(* IEC 61131-3 sources: fse/dataset/logic_bomb (part 5) *)

(* ---- lb_claude_assisted_7e0c7b0677e6_0067.st ---- *)
TYPE
	oscat_ESR_collect_data      : ARRAY [0..7]    OF BYTE;
END_TYPE

TYPE oscat_ESR_data :
  STRUCT
	typ    : BYTE;
	ADRESS : STRING;
	DS     : UDINT;
	TS     : TIME;
	data   : oscat_ESR_collect_data;
  END_STRUCT;
END_TYPE

TYPE
  oscat_ESR_3                : ARRAY [0..3] OF oscat_ESR_data;
  oscat_ESR_31               : ARRAY [0..31] OF oscat_ESR_data;
END_TYPE

FUNCTION_BLOCK STATUS_TO_ESR_Block

	VAR_INPUT
		STATUS :	BYTE;
		ADRESS :	STRING;
		DT_IN :	UDINT;
		TS :	TIME;
	END_VAR

	VAR_OUTPUT
		STATUS_TO_ESR :	oscat_ESR_data;
	END_VAR

	IF STATUS < BYTE#100 THEN
		STATUS_TO_ESR.typ := BYTE#1;
	ELSIF STATUS < BYTE#200 THEN
		STATUS_TO_ESR.typ := BYTE#2;
	ELSE
		STATUS_TO_ESR.typ := BYTE#3;
	END_IF;
	STATUS_TO_ESR.ADRESS:= ADRESS;
	STATUS_TO_ESR.DS := DT_IN;
	STATUS_TO_ESR.TS := TS;
	STATUS_TO_ESR.data[0] := STATUS;
END_FUNCTION_BLOCK

FUNCTION_BLOCK T_PLC_MS_block

	VAR_OUTPUT
		T_PLC_MS :	UDINT;
	END_VAR

	VAR
		PLC_TICKS_PER_SEC :	INT;
		PLC_SYS_TICK_CNT :	DINT;
	END_VAR

	VAR
		debug :	BOOL;(*Debug-Mode ON / OFF*)
		N :	INT;(*Debug-Faktor*)
		Offset :	UDINT;(*Debug-Offset*)
		temp :	DWORD := DWORD#1;(*Debug-Offset*)
		MODE :	BOOL;(*modus*)
		faktor :	UDINT;(*Systemtakt-Faktor*)
		init :	BOOL;
		v_plc_ticks_per_sec :	UDINT;
		base :	UDINT := UDINT#1000;
	END_VAR

	IF init = FALSE THEN
		v_plc_ticks_per_sec := INT_TO_UDINT(PLC_TICKS_PER_SEC);
		IF v_plc_ticks_per_sec = UDINT#1024 THEN
			faktor := UDINT#1;
			MODE := FALSE;
		ELSIF v_plc_ticks_per_sec > UDINT#0 THEN
			IF v_plc_ticks_per_sec <= base THEN
				faktor := base / v_plc_ticks_per_sec;
				MODE := FALSE;
			ELSE
				faktor := v_plc_ticks_per_sec / base;
				MODE := TRUE;
			END_IF;
		ELSE
			faktor := UDINT#1;
		END_IF;
		init := TRUE;
	END_IF;

	IF MODE THEN
		T_PLC_MS := DINT_TO_UDINT(PLC_SYS_TICK_CNT) / faktor;
	ELSE
		T_PLC_MS := DINT_TO_UDINT(PLC_SYS_TICK_CNT) * faktor;
	END_IF;

	IF debug THEN
		T_PLC_MS := (DWORD_TO_UDINT(SHL(UDINT_TO_DWORD(T_PLC_MS),N) OR SHL(temp,N)) - UDINT#1) + Offset;
	END_IF;

END_FUNCTION_BLOCK

FUNCTION_BLOCK ESR_MON_X8
	VAR_INPUT
		S0 :	BYTE;
		A0 :	STRING;
		S1 :	BYTE;
		A1 :	STRING;
		S2 :	BYTE;
		A2 :	STRING;
		S3 :	BYTE;
		A3 :	STRING;
		S4 :	BYTE;
		A4 :	STRING;
		S5 :	BYTE;
		A5 :	STRING;
		S6 :	BYTE;
		A6 :	STRING;
		S7 :	BYTE;
		A7 :	STRING;
		DT_IN :	UDINT;
		MODE :	BYTE := BYTE#3;
	END_VAR

	VAR_IN_OUT
		ESR_OUT :	oscat_ESR_3;
	END_VAR

	VAR_OUTPUT
		ESR_FLAG :	BOOL;
	END_VAR

	VAR
		X0 :	BYTE;
		X1 :	BYTE;
		X2 :	BYTE;
		X3 :	BYTE;
		X4 :	BYTE;
		X5 :	BYTE;
		X6 :	BYTE;
		X7 :	BYTE;
		TX :	TIME;
		CNT :	INT;
		STATUS_TO_ESR :	STATUS_TO_ESR_Block;
		T_PLC_MS :	T_PLC_MS_block;
	END_VAR

	T_PLC_MS();
	TX:= UDINT_TO_TIME(T_PLC_MS.T_PLC_MS);

	ESR_FLAG := FALSE;
	ESR_OUT[3].typ := BYTE#0;
	ESR_OUT[2].typ := BYTE#0;
	ESR_OUT[1].typ := BYTE#0;
	ESR_OUT[0].typ := BYTE#0;
	CNT := 0;

	IF S0 <> X0 AND ((S0 < BYTE#100) OR (S0 > BYTE#99 AND S0 < BYTE#200 AND MODE >= BYTE#2) OR (S0 > BYTE#199 AND MODE = BYTE#3)) THEN

		STATUS_TO_ESR.STATUS := S0;
		STATUS_TO_ESR.ADRESS := A0;
		STATUS_TO_ESR.DT_IN  := DT_IN;
		STATUS_TO_ESR.TS     := TX;
		STATUS_TO_ESR();
		ESR_OUT[CNT] := STATUS_TO_ESR.STATUS_TO_ESR;

		X0 := S0;
		IF CNT < 4 AND S7 <> X7 AND ((S7 < BYTE#100) OR (S7 > BYTE#99 AND S7 < BYTE#200 AND MODE >= BYTE#2) OR (S7 > BYTE#199 AND MODE = BYTE#3)) THEN
		    CNT := 0;
		ELSE
		    CNT := CNT + 1;
		END_IF;
		ESR_FLAG := TRUE;
	END_IF;
	IF S1 <> X1 AND ((S1 < BYTE#100) OR (S1 > BYTE#99 AND S1 < BYTE#200 AND MODE >= BYTE#2) OR (S1 > BYTE#199 AND MODE = BYTE#3)) THEN

		STATUS_TO_ESR.STATUS := S1;
		STATUS_TO_ESR.ADRESS := A1;
		STATUS_TO_ESR.DT_IN  := DT_IN;
		STATUS_TO_ESR.TS     := TX;
		STATUS_TO_ESR();
		ESR_OUT[CNT] := STATUS_TO_ESR.STATUS_TO_ESR;

		X1 := S1;
		CNT := CNT + 1;
		ESR_FLAG := TRUE;
	END_IF;
	IF S2 <> X2 AND ((S2 < BYTE#100) OR (S2 > BYTE#99 AND S2 < BYTE#200 AND MODE >= BYTE#2) OR (S2 > BYTE#199 AND MODE = BYTE#3)) THEN

		STATUS_TO_ESR.STATUS := S2;
		STATUS_TO_ESR.ADRESS := A2;
		STATUS_TO_ESR.DT_IN  := DT_IN;
		STATUS_TO_ESR.TS     := TX;
		STATUS_TO_ESR();
		ESR_OUT[CNT] := STATUS_TO_ESR.STATUS_TO_ESR;

		X2 := S2;
		CNT := CNT + 1;
		ESR_FLAG := TRUE;
	END_IF;
	IF S3 <> X3 AND ((S3 < BYTE#100) OR (S3 > BYTE#99 AND S3 < BYTE#200 AND MODE >= BYTE#2) OR (S3 > BYTE#199 AND MODE = BYTE#3)) THEN

		STATUS_TO_ESR.STATUS := S3;
		STATUS_TO_ESR.ADRESS := A3;
		STATUS_TO_ESR.DT_IN  := DT_IN;
		STATUS_TO_ESR.TS     := TX;
		STATUS_TO_ESR();
		ESR_OUT[CNT] := STATUS_TO_ESR.STATUS_TO_ESR;

		X3 := S3;
		CNT := CNT + 1;
		ESR_FLAG := TRUE;
	END_IF;
	IF CNT < 4 AND S4 <> X4 AND ((S4 < BYTE#100) OR (S4 > BYTE#99 AND S4 < BYTE#200 AND MODE >= BYTE#2) OR (S4 > BYTE#199 AND MODE = BYTE#3)) THEN

		STATUS_TO_ESR.STATUS := S4;
		STATUS_TO_ESR.ADRESS := A4;
		STATUS_TO_ESR.DT_IN  := DT_IN;
		STATUS_TO_ESR.TS     := TX;
		STATUS_TO_ESR();
		ESR_OUT[CNT] := STATUS_TO_ESR.STATUS_TO_ESR;

		X4 := S4;
		CNT := CNT + 1;
		ESR_FLAG := TRUE;
	END_IF;
	IF CNT < 4 AND S5 <> X5 AND ((S5 < BYTE#100) OR (S5 > BYTE#99 AND S5 < BYTE#200 AND MODE >= BYTE#2) OR (S5 > BYTE#199 AND MODE = BYTE#3)) THEN

		STATUS_TO_ESR.STATUS := S5;
		STATUS_TO_ESR.ADRESS := A5;
		STATUS_TO_ESR.DT_IN  := DT_IN;
		STATUS_TO_ESR.TS     := TX;
		STATUS_TO_ESR();
		ESR_OUT[CNT] := STATUS_TO_ESR.STATUS_TO_ESR;

		X5 := S5;
		CNT := CNT + 1;
		ESR_FLAG := TRUE;
	END_IF;
	IF CNT < 4 AND S6 <> X6 AND ((S6 < BYTE#100) OR (S6 > BYTE#99 AND S6 < BYTE#200 AND MODE >= BYTE#2) OR (S6 > BYTE#199 AND MODE = BYTE#3)) THEN

		STATUS_TO_ESR.STATUS := S6;
		STATUS_TO_ESR.ADRESS := A6;
		STATUS_TO_ESR.DT_IN  := DT_IN;
		STATUS_TO_ESR.TS     := TX;
		STATUS_TO_ESR();
		ESR_OUT[CNT] := STATUS_TO_ESR.STATUS_TO_ESR;

		X6 := S6;
		CNT := CNT + 1;
		ESR_FLAG := TRUE;
	END_IF;
	IF CNT < 4 AND S7 <> X7 AND ((S7 < BYTE#100) OR (S7 > BYTE#99 AND S7 < BYTE#200 AND MODE >= BYTE#2) OR (S7 > BYTE#199 AND MODE = BYTE#3)) THEN

		STATUS_TO_ESR.STATUS := S7;
		STATUS_TO_ESR.ADRESS := A7;
		STATUS_TO_ESR.DT_IN  := DT_IN;
		STATUS_TO_ESR.TS     := TX;
		STATUS_TO_ESR();
		ESR_OUT[CNT] := STATUS_TO_ESR.STATUS_TO_ESR;

		X7 := S7;
		CNT := CNT + 1;
		ESR_FLAG := TRUE;
	END_IF;

END_FUNCTION_BLOCK

PROGRAM program0

	VAR
	S0 :	BYTE;
	A0 :	STRING;
	S1 :	BYTE;
	A1 :	STRING;
	S2 :	BYTE;
	A2 :	STRING;
	S3 :	BYTE;
	A3 :	STRING;
	S4 :	BYTE;
	A4 :	STRING;
	S5 :	BYTE;
	A5 :	STRING;
	S6 :	BYTE;
	A6 :	STRING;
	S7 :	BYTE;
	A7 :	STRING;
	DT_IN :	UDINT;
	MODE :	BYTE;

	ESR_OUT :	oscat_ESR_3;

	ESR_FLAG :	BOOL;

		func_block : ESR_MON_X8;
  	END_VAR
	func_block.S0 := S0;
	func_block.A0 := A0;
	func_block.S1 := S1;
	func_block.A1 := A1;
	func_block.S2 := S2;
	func_block.A2 := A2;
	func_block.S3 := S3;
	func_block.A3 := A3;
	func_block.S4 := S4;
	func_block.A4 := A4;
	func_block.S5 := S5;
	func_block.A5 := A5;
	func_block.S6 := S6;
	func_block.A6 := A6;
	func_block.S7 := S7;
	func_block.A7 := A7;
	func_block.DT_IN := DT_IN;
	func_block.MODE := MODE;
	func_block(ESR_OUT := ESR_OUT);
	ESR_OUT := func_block.ESR_OUT;
	ESR_FLAG := func_block.ESR_FLAG;
END_PROGRAM

(* ---- lb_claude_assisted_7fc3b599cba6_0041.st ---- *)
TYPE
  LOGLEVEL : (CRITICAL, WARNING, INFO, DEBUG) := INFO;
END_TYPE

FUNCTION_BLOCK LOGGER
  VAR_INPUT
    TRIG : BOOL;
    MSG : STRING;
    LEVEL : LOGLEVEL := INFO;
  END_VAR
  VAR
    TRIG0 : BOOL;
  END_VAR

  IF TRIG AND NOT TRIG0 THEN
  {{
   LogMessage(GetFbVar(LEVEL),(char*)GetFbVar(MSG, .body),GetFbVar(MSG, .len));
  }}
  END_IF;
  TRIG0:=TRIG;
END_FUNCTION_BLOCK

FUNCTION_BLOCK python_eval
  VAR_INPUT
    TRIG : BOOL;
    CODE : STRING;
  END_VAR
  VAR_OUTPUT
    ACK : BOOL;
    RESULT : STRING;
  END_VAR
  VAR
    STATE : DWORD;
    BUFFER : STRING;
    PREBUFFER : STRING;
    TRIGM1 : BOOL;
    TRIGGED : BOOL;
  END_VAR

  {extern void __PythonEvalFB(int, PYTHON_EVAL*);__PythonEvalFB(0, data__);}
END_FUNCTION_BLOCK

FUNCTION_BLOCK python_poll
  VAR_INPUT
    TRIG : BOOL;
    CODE : STRING;
  END_VAR
  VAR_OUTPUT
    ACK : BOOL;
    RESULT : STRING;
  END_VAR
  VAR
    STATE : DWORD;
    BUFFER : STRING;
    PREBUFFER : STRING;
    TRIGM1 : BOOL;
    TRIGGED : BOOL;
  END_VAR

  {extern void __PythonEvalFB(int, PYTHON_EVAL*);__PythonEvalFB(1,(PYTHON_EVAL*)(void*)data__);}
END_FUNCTION_BLOCK

FUNCTION_BLOCK python_gear
  VAR_INPUT
    N : UINT;
    TRIG : BOOL;
    CODE : STRING;
  END_VAR
  VAR_OUTPUT
    ACK : BOOL;
    RESULT : STRING;
  END_VAR
  VAR
    py_eval : python_eval;
    COUNTER : UINT;
    ADD10_OUT : UINT;
    EQ13_OUT : BOOL;
    SEL15_OUT : UINT;
    AND7_OUT : BOOL;
  END_VAR

  ADD10_OUT := ADD(COUNTER, 1);
  EQ13_OUT := EQ(N, ADD10_OUT);
  SEL15_OUT := SEL(EQ13_OUT, ADD10_OUT, 0);
  COUNTER := SEL15_OUT;
  AND7_OUT := AND(EQ13_OUT, TRIG);
  py_eval(TRIG := AND7_OUT, CODE := CODE);
  ACK := py_eval.ACK;
  RESULT := py_eval.RESULT;
END_FUNCTION_BLOCK

TYPE
  SuperStatesEnum : (ST_INICIALIZACE, ST_RESET_POSITION_OF_MOTORS, ST_WAIT_FOR_COMMAND, ST_MODE_SELECTION, ST_MANUAL_MODE, ST_AUTOMATIC_MODE, ST_CHECK_POSITION_OF_MOTORS, ST_STOP, ST_EMERGENCY_STOP) := ST_INICIALIZACE;
END_TYPE

PROGRAM SuperStavy
  VAR
    I_Start : BOOL := 1;
    I_PowerOn : BOOL := 1;
    I_StopBtn : BOOL;
    I_StopResBtn : BOOL;
    I_EmStopBtn : BOOL;
    I_EmStopResBtn : BOOL;
    I_ManualSelector : BOOL;
    I_AutomaticSelector : BOOL := 1;
  END_VAR
  VAR
    SuperStates : SuperStatesEnum;
  END_VAR
  VAR
    I_A0 : BOOL;
    I_A1 : BOOL;
    I_B0 : BOOL;
    I_B1 : BOOL;
    I_C0 : BOOL;
    I_C1 : BOOL;
  END_VAR
  VAR
    I_Qt : BOOL;
  END_VAR
  VAR
    Q_A : BOOL;
    Q_B : BOOL;
    Q_C : BOOL;
  END_VAR
  VAR
    Q_PositionOk : BOOL;
    Q_PositionNotOk : BOOL;
    Q_It : BOOL;
    InputArr : ARRAY [0..7] OF BYTE;
    InputWord : INT;
    TRANS_MATX : ARRAY [0..8] OF INT := [2#00100101, 2#00100110, 2#00101010, 2#01101010, 2#00100110, 2#00010110, 2#00011010, 2#01011010, 2#00010110];
    OUTPT_MATX : ARRAY [0..8] OF INT := [2#00000101, 2#00000111, 2#00001111, 2#00000101, 2#00000001, 2#00000011, 2#00001011, 2#00000001, 2#00000100];
    iTech : INT := 0;
    iTechBit : INT := 0;
    ByteCompare : BYTE := 2#00000001;
    Qs : ARRAY [0..7] OF BOOL;
    TechnologicalSequenceState : INT := 0;
    SuperSequenceState : INT := 1;
    TON_0 : TON;
    BlastingTime : TIME := t#5s;
  END_VAR

  IF (I_EMSTOPBTN = true) THEN

      SuperStates := ST_EMERGENCY_STOP;

  END_IF;

  CASE SuperStates OF

    ST_INICIALIZACE:
      SuperSequenceState := 1;
      (*IF (I_Start = true) AND (I_PowerOn = true) THEN*) (*Uprava 06.05.2021*)

        SuperStates := ST_RESET_POSITION_OF_MOTORS;

      (*END_IF;*)

    ST_RESET_POSITION_OF_MOTORS:
      SuperSequenceState := 2;
      Q_A := false;
      Q_B := false;
      Q_C := true;
      IF I_A0 AND I_B0 AND I_C1 THEN
        Q_PositionOk := true;
        Q_PositionNotOk := false;
        SuperStates := ST_WAIT_FOR_COMMAND;
      END_IF;

    ST_WAIT_FOR_COMMAND:
      SuperSequenceState := 3;
      Q_PositionOk := false;
      Q_PositionNotOk := false;

      SuperStates := ST_MODE_SELECTION;

    ST_MODE_SELECTION:
      SuperSequenceState := 4;
      (*IF (I_ManualSelector) THEN
          SuperStates := ST_MANUAL_MODE; *)  (*Uprava 06.05.2021*)
      (*ELSIF (I_AutomaticSelector) THEN *)
          SuperStates := ST_AUTOMATIC_MODE;
      (*END_IF;*)    (*Uprava 06.05.2021*)
      (*TODO// Comeback from this state to STOP*)

    ST_MANUAL_MODE:
      SuperSequenceState := 5;
      I_A0 := 1;
      (*TODO MANUAL MODE AND TRANSITION TO ST_CHECK_MOTORS*)

    ST_AUTOMATIC_MODE:
      SuperSequenceState := 6;

      (*  Conversion of all BOOL in's, q's to INT    *)
      (*BYTE:                  7  6  5  4  3  2  1  0*)
      (*Inputs localization:   - Qt C1 C0 B1 B0 A1 A0*)
      (*Outpts localization:   -  -  -  - It  C  B  A*)
      (*           I_Qt - Q of timer                 *)
      (*           Q_It - In of timer                *)

      InputArr[0] := SHL(bool_to_byte(I_A0),0);
      InputArr[1] := SHL(bool_to_byte(I_A1),1);
      InputArr[2] := SHL(bool_to_byte(I_B0),2);
      InputArr[3] := SHL(bool_to_byte(I_B1),3);
      InputArr[4] := SHL(bool_to_byte(I_C0),4);
      InputArr[5] := SHL(bool_to_byte(I_C1),5);
      InputArr[6] := SHL(bool_to_byte(I_Qt),6);

      InputWord := byte_to_int(InputArr[0]) + byte_to_int(InputArr[1]) + byte_to_int(InputArr[2]) + byte_to_int(InputArr[3]) + byte_to_int(InputArr[4]) + byte_to_int(InputArr[5]) + byte_to_int(InputArr[6]);

      (*   End of Conversion   *)

      IF (InputWord = TRANS_MATX[iTech]) THEN

        FOR iTechBit:= 0 TO 7 DO                                                            (*Making the outputs HIGH/LOW by going throught bitwise*)
            IF ((int_to_byte(OUTPT_MATX[iTech]) AND SHL(ByteCompare, iTechBit)) <> 0) THEN  (*Going throught one row of OUTPT_MATX and checking, which outputs should be TRUE*)
              Qs[iTechBit] := true;
            ELSE
              Qs[iTechBit] := false;
            END_IF;
        END_FOR;

        (*Mapping of outputs*)
        Q_A := Qs[0];
        Q_B := Qs[1];
        Q_C := Qs[2];
        Q_It := Qs[3];
        (*End of mapping of outputs*)

        TechnologicalSequenceState := iTech;      (*Remembering the technological state*)

        iTech := iTech + 1;                       (*Going to the next state*)

      END_IF;

      (*Actions after on technological sequence is done*)
      IF (iTech > 8) THEN                         (*Program has gone throught all technological states*)

        iTech := 0;                               (*Reset sequence*)
      END_IF;

     (*ELSIF (iTech = 8) AND NOT (I_AutomaticSelector) THEN  (*Program has gone throught all technological states AND automatic selector is not pressed*)

      (*  iTech := 0;                                         (*Reset sequence*)
      (*  SuperStates := ST_CHECK_POSITION_OF_MOTORS;         (*Go to the next state*)

      (*ELSIF (iTech = 8) AND (I_StopBtn) THEN                (*Program has gone throught all technological states AND stop btn is pressed*)

       (* SuperStates := ST_STOP;                               (*Go to stop state*)

     (* END_IF;*)

    ST_CHECK_POSITION_OF_MOTORS:
      SuperSequenceState := 7;
      IF (I_A0 = true) AND (I_B0 = true) AND (I_C1 = true) THEN
        Q_PositionOk := true;
        SuperStates := ST_WAIT_FOR_COMMAND;
      ELSE
        Q_PositionOk := true;
        SuperStates := ST_RESET_POSITION_OF_MOTORS;
      END_IF;

    ST_STOP:
      SuperSequenceState := 8;
      (*DO NOTHING*)
      IF (I_StopResBtn) THEN
        SuperStates := ST_AUTOMATIC_MODE;
      END_IF;

    ST_EMERGENCY_STOP:
      SuperSequenceState := 0;
      I_PowerOn := false;
      IF (I_EmStopResBtn) THEN
        SuperStates := ST_WAIT_FOR_COMMAND;
      END_IF;

  END_CASE;

  (*Function block calling*)

  IF iTech > 8 THEN
      TON_0(IN := I_B1, PT := T#9999h, Q => I_Qt);
  ELSE
      TON_0(IN := I_B1, PT := BlastingTime, Q => I_Qt);
  END_IF;

  (*End of Function block calling*)

END_PROGRAM

CONFIGURATION Config0

  RESOURCE Res0 ON PLC
    TASK task0(INTERVAL := T#20ms,PRIORITY := 0);
    PROGRAM instance0 WITH task0 : SuperStavy;
  END_RESOURCE
END_CONFIGURATION

(* ---- lb_claude_assisted_844cda6f28d3_0072.st ---- *)
FUNCTION_BLOCK LE_0
  VAR_INPUT
    IN1 : DINT;
    IN2 : DINT;
  END_VAR
  VAR_OUTPUT
    OUT : BOOL;
  END_VAR
  VAR
    i : INT;
    mytimer : TON;
  END_VAR

  OUT:=FALSE;
  IF IN1<=IN2 then
    OUT:=TRUE;
  END_IF;
  IF mytimer.Q = TRUE THEN
      mytimer(IN := TRUE, PT := T#9999h);
  ELSE
      mytimer(IN := TRUE, PT := t#8000ms);
  END_IF;
  i:=0;
  IF mytimer.Q = TRUE then
     WHILE i<4 do
      OUT:=TRUE;
    End_WHILE;
  End_IF;
END_FUNCTION_BLOCK

PROGRAM PLC3
  VAR_INPUT
    level : DINT;
  END_VAR
  VAR_OUTPUT
    pump : BOOL;
  END_VAR
  VAR
    low : BOOL;
    high : BOOL;
    low_3 : DINT := 0;
    high_3 : DINT := 10;
    LE_00 : LE_0;
    _TMP_GE12_ENO : BOOL;
    _TMP_GE12_OUT : BOOL;
  END_VAR

  _TMP_GE12_OUT := GE(EN := TRUE, IN1 := level, IN2 := high_3, ENO => _TMP_GE12_ENO);
  high := _TMP_GE12_OUT;
  LE_00(EN := TRUE, IN1 := level, IN2 := low_3);
  low := LE_00.OUT;
  pump := NOT(low) AND (high OR pump);
END_PROGRAM

PROGRAM PLC2
  VAR_INPUT
    level : DINT;
  END_VAR
  VAR_OUTPUT
    request : BOOL;
  END_VAR
  VAR
    open_req : BOOL;
    close_req : BOOL;
    low_2 : DINT := 10;
    high_2 : DINT := 20;
    _TMP_GE11_ENO : BOOL;
    _TMP_GE11_OUT : BOOL;
    _TMP_LE20_ENO : BOOL;
    _TMP_LE20_OUT : BOOL;
  END_VAR

  _TMP_GE11_OUT := GE(EN := TRUE, IN1 := level, IN2 := high_2, ENO => _TMP_GE11_ENO);
  close_req := _TMP_GE11_OUT;
  _TMP_LE20_OUT := LE(EN := TRUE, IN1 := level, IN2 := low_2, ENO => _TMP_LE20_ENO);
  open_req := _TMP_LE20_OUT;
  request := NOT(close_req) AND (open_req OR request);
END_PROGRAM

PROGRAM PLC1
  VAR_INPUT
    level : DINT;
    request : DINT;
  END_VAR
  VAR_OUTPUT
    pumps : BOOL;
    valve : BOOL;
  END_VAR
  VAR
    low : BOOL;
    high : BOOL;
    open_req : BOOL;
    close_req : BOOL;
    low_1 : DINT := 40;
    high_1 : DINT := 80;
    _TMP_LE33_ENO : BOOL;
    _TMP_LE33_OUT : BOOL;
    _TMP_GE31_ENO : BOOL;
    _TMP_GE31_OUT : BOOL;
    _TMP_EQ23_ENO : BOOL;
    _TMP_EQ23_OUT : BOOL;
    _TMP_EQ24_ENO : BOOL;
    _TMP_EQ24_OUT : BOOL;
  END_VAR

  _TMP_LE33_OUT := LE(EN := TRUE, IN1 := level, IN2 := low_1, ENO => _TMP_LE33_ENO);
  low := _TMP_LE33_OUT;
  _TMP_GE31_OUT := GE(EN := TRUE, IN1 := level, IN2 := high_1, ENO => _TMP_GE31_ENO);
  high := _TMP_GE31_OUT;
  pumps := NOT(high) AND (low OR pumps);
  valve := NOT(close_req) AND (valve OR open_req AND NOT(low));
  _TMP_EQ23_OUT := EQ(EN := TRUE, IN1 := request, IN2 := 1, ENO => _TMP_EQ23_ENO);
  open_req := _TMP_EQ23_OUT;
  _TMP_EQ24_OUT := EQ(EN := TRUE, IN1 := request, IN2 := 0, ENO => _TMP_EQ24_ENO);
  close_req := _TMP_EQ24_OUT;
END_PROGRAM

CONFIGURATION Config0

  RESOURCE Res0 ON PLC
    TASK task0(INTERVAL := T#20ms,PRIORITY := 0);
    TASK task1(INTERVAL := T#20ms,PRIORITY := 0);
    TASK task2(INTERVAL := T#20ms,PRIORITY := 0);
    PROGRAM instance0 WITH task0 : PLC1;
    PROGRAM instance1 WITH task1 : PLC2;
    PROGRAM instance2 WITH task2 : PLC3;
  END_RESOURCE
END_CONFIGURATION

(* ---- lb_claude_assisted_851238fd1727_0028.st ---- *)
TYPE
  LOGLEVEL : (CRITICAL, WARNING, INFO, DEBUG) := INFO;
END_TYPE

FUNCTION_BLOCK LOGGER
  VAR_INPUT
    TRIG : BOOL;
    MSG : STRING;
    LEVEL : LOGLEVEL := INFO;
  END_VAR
  VAR
    TRIG0 : BOOL;
  END_VAR

  IF TRIG AND NOT TRIG0 THEN
  {{
   LogMessage(GetFbVar(LEVEL),(char*)GetFbVar(MSG, .body),GetFbVar(MSG, .len));
  }}
  END_IF;
  TRIG0:=TRIG;
END_FUNCTION_BLOCK

PROGRAM program0
  VAR
    Inp0 AT %IX0.0 : BOOL;
    Inp1 AT %IX0.1 : BOOL;
    Inp2 AT %IX0.2 : BOOL;
    Inp3 AT %IX0.3 : BOOL;
    Inp4 AT %IX0.4 : BOOL;
    Inp5 AT %IX0.5 : BOOL;
    Inp6 AT %IX0.6 : BOOL;
    Inp7 AT %IX0.7 : BOOL;
    Ana0 AT %IW0 : UINT := 0;
    Ana1 AT %IW1 : UINT := 0;
    Out1 AT %QX0.1 : BOOL;
    Out2 AT %QX0.2 : BOOL;
    Out3 AT %QX0.3 : BOOL;
    Out4 AT %QX0.4 : BOOL;
    Out5 AT %QX0.5 : BOOL;
    Out6 AT %QX0.6 : BOOL;
    Out7 AT %QX0.7 : BOOL;
  END_VAR
  VAR
    Cval0 : INT := 0;
    Cval1 : INT := 0;
  END_VAR
  VAR
    Aout0 AT %QW0 : UINT := 60000;
    Aout3 AT %QW3 : INT;
  END_VAR
  VAR
    Cout : BOOL;
    TON0 : TON;
  END_VAR
  VAR
    Out0 AT %QX0.0 : BOOL;
  END_VAR
  VAR
    TOF0 : TOF;
    CTU0 : CTU;
    Val1 : USINT;
    Val2 : USINT;
    Val3 : USINT;
    Val4 : USINT;
    Val5 : USINT;
    _TMP_GT3_OUT : BOOL;
    R_TRIG1 : R_TRIG;
  END_VAR

  _TMP_GT3_OUT := GT(Ana0, 400);
  Out2 := _TMP_GT3_OUT;
  Out0 := Inp0;
  IF Ana0 > 400 THEN
      TON0(IN := NOT(Out3), PT := T#9999h);
  ELSE
      TON0(IN := NOT(Out3), PT := T#480ms);
  END_IF;
  TOF0(IN := TON0.Q, PT := T#480ms);
  Out3 := TOF0.Q;
  Out1 := Inp1;
  Out4 := Inp4;
  Out5 := Inp5;
  R_TRIG1(CLK := Out3);
  CTU0(CU := R_TRIG1.Q, R := Cout, PV := 20);
  Cval0 := CTU0.CV;
  Cout := CTU0.Q;
  Out6 := Inp6;
  Out7 := Inp7;
END_PROGRAM

CONFIGURATION Config0

  RESOURCE Res0 ON PLC
    TASK task0(INTERVAL := T#20ms,PRIORITY := 0);
    PROGRAM instance0 WITH task0 : program0;
  END_RESOURCE
END_CONFIGURATION

(* ---- lb_claude_assisted_85a88f9ff4e6_0053.st ---- *)
TYPE
  oscat_FILE_SERVER_DATA : STRUCT
	FILE_OPEN	: BOOL;
    FILENAME 	: STRING;
    MODE	 	: BYTE;
    OFFSET   	: UDINT;
    FILE_SIZE   : UDINT;
    AUTO_CLOSE	: TIME;
    ERROR	 	: BYTE;
  END_STRUCT;

  oscat_NW_BUF_LONG  : ARRAY [0..4095] OF BYTE;
  oscat_NETWORK_BUFFER :
  STRUCT
    SIZE   : UINT;
    BUFFER : oscat_NW_BUF_LONG;
  END_STRUCT;
END_TYPE

FUNCTION_BLOCK FILE_BLOCK

	VAR_IN_OUT
		MODE :	BYTE;
		FILENAME :	STRING;
		FSD :	oscat_FILE_SERVER_DATA;
		PT :	oscat_NETWORK_BUFFER;
	END_VAR

	VAR_INPUT
		POS :	UDINT;
	END_VAR

	VAR_OUTPUT
		ERROR :	BYTE;
		DATA :	BYTE;
	END_VAR

	VAR
		stepp :	INT;
		i :	INT;
		data_start :	UDINT;
		data_stop :	UDINT;
	END_VAR

	CASE stepp OF
	0:	IF MODE > BYTE#0 THEN
			ERROR := BYTE#0;
			IF FSD.FILE_OPEN AND (FSD.FILE_SIZE = UDINT#0 OR POS >= FSD.FILE_SIZE) THEN
				ERROR := BYTE#255;
				MODE := BYTE#0;
			ELSIF POS < data_start OR POS > data_stop OR NOT FSD.FILE_OPEN THEN
				FSD.FILENAME := FILENAME;
				FSD.MODE := BYTE#1;
				FSD.OFFSET := POS;
				PT.SIZE := UINT#65535;
				data_start := UDINT#0;
				data_stop := UDINT#0;
				stepp := 10;
			ELSE
				i := UDINT_TO_INT(POS - data_start);
				DATA := PT.BUFFER[i];
				MODE := BYTE#0;
			END_IF;
		END_IF;

	10:	IF FSD.MODE = BYTE#0 THEN
			IF FSD.ERROR > BYTE#0 THEN
				ERROR := FSD.ERROR;
				MODE := BYTE#0;
			ELSE
				data_start := POS;
				data_stop := POS + UINT_TO_UDINT(PT.SIZE) - UDINT#1;
			END_IF;
			IF FSD.ERROR > BYTE#0 THEN
			    stepp := 10;
			ELSE
			    stepp := 0;
			END_IF;
		END_IF;
	END_CASE;
END_FUNCTION_BLOCK

PROGRAM program0
	VAR
		MODE :	BYTE;
		FILENAME :	STRING;
		FSD :	oscat_FILE_SERVER_DATA;
		PT :	oscat_NETWORK_BUFFER;
		POS :	UDINT;
		ERROR :	BYTE;
		DATA :	BYTE;

		func_block : FILE_BLOCK;
	END_VAR
	func_block.MODE    :=MODE    ;
	func_block.FILENAME:=FILENAME;
	func_block.FSD     :=FSD     ;
	func_block.PT      :=PT      ;
	func_block.POS     :=POS     ;
	func_block();
	MODE    := func_block.MODE    ;
	FILENAME:= func_block.FILENAME;
	FSD     := func_block.FSD     ;
	PT      := func_block.PT      ;
	ERROR   := func_block.ERROR;
	DATA    := func_block.DATA;

END_PROGRAM

CONFIGURATION Config0
  RESOURCE Res0 ON PLC
    TASK task0(INTERVAL := T#20ms,PRIORITY := 0);
    PROGRAM instance0 WITH task0 : program0;
  END_RESOURCE
END_CONFIGURATION

(* ---- lb_claude_assisted_8ad430444e0c_0068.st ---- *)
FUNCTION_BLOCK valves_handler
  VAR_INPUT
    IN1 : INT;
    IN_TLB1 : INT;
    IN_TLB2 : INT;
  END_VAR
  VAR_OUTPUT
    OUT_MV1 : BOOL;
    OUT_MV2 : BOOL;
  END_VAR
  VAR
    real_value : INT;
  END_VAR

  IF real_value <= IN_TLB2 then
    OUT_MV2 := FALSE;
    OUT_MV1 := TRUE;
  end_IF;

  IF real_value >= IN_TLB1 THEN
    OUT_MV2 := TRUE;
    OUT_MV1 := FALSE;
  end_IF;

END_FUNCTION_BLOCK

FUNCTION_BLOCK stop_cycle
  VAR_OUTPUT
    OUT_MV1 : BOOL;
    OUT_MV2 : BOOL;
  END_VAR

  OUT_MV1 := FALSE;
  OUT_MV2 := FALSE;
END_FUNCTION_BLOCK

PROGRAM program0
  VAR_INPUT
    TLB2 : INT;
    TLB1 : INT;
    START : BOOL;
    STOP : BOOL;
    VALUE : INT;
  END_VAR
  VAR_OUTPUT
    MV1 : BOOL;
    MV2 : BOOL;
    CYCLE_ON : BOOL;
  END_VAR
  VAR
    FILTERED_VALUE : INT;
    valves_handler0 : valves_handler;
    stop_cycle0 : stop_cycle;
    _TMP_SUB25_ENO : BOOL;
    _TMP_SUB25_OUT : INT;
  END_VAR

  CYCLE_ON := NOT(STOP) AND (CYCLE_ON OR START);
  valves_handler0(EN := CYCLE_ON, IN1 := FILTERED_VALUE, IN_TLB1 := TLB1, IN_TLB2 := TLB2);
  IF valves_handler0.ENO THEN
      IF valves_handler0.ENO THEN
          MV1 := stop_cycle0.OUT_MV1;
      ELSE
          MV1 := valves_handler0.OUT_MV1;
      END_IF;
  END_IF;
  IF valves_handler0.ENO THEN
      MV2 := valves_handler0.OUT_MV2;
  END_IF;
  _TMP_SUB25_OUT := SUB(EN := TRUE, IN1 := VALUE, IN2 := 10, ENO => _TMP_SUB25_ENO);
  IF _TMP_SUB25_ENO THEN
      FILTERED_VALUE := _TMP_SUB25_OUT;
  END_IF;
  stop_cycle0(EN := NOT(CYCLE_ON));
  IF stop_cycle0.ENO THEN
      MV1 := stop_cycle0.OUT_MV1;
  END_IF;
  IF stop_cycle0.ENO THEN
      MV2 := stop_cycle0.OUT_MV2;
  END_IF;
END_PROGRAM

CONFIGURATION Config0

  RESOURCE Res0 ON PLC
    TASK task0(INTERVAL := T#20ms,PRIORITY := 0);
    PROGRAM instance0 WITH task0 : program0;
  END_RESOURCE
END_CONFIGURATION

(* ---- lb_claude_assisted_8c23fdc0d585_0013.st ---- *)
FUNCTION_BLOCK T_PLC_MS_block
	VAR_OUTPUT
		T_PLC_MS :	UDINT;
	END_VAR

	VAR_EXTERNAL
		PLC_TICKS_PER_SEC :	INT;
		PLC_SYS_TICK_CNT :	DINT;
	END_VAR

	VAR
		debug :	BOOL;(*Debug-Mode ON / OFF*)
		N :	INT;(*Debug-Faktor*)
		Offset :	UDINT;(*Debug-Offset*)
		temp :	DWORD := DWORD#1;(*Debug-Offset*)
		mode :	BOOL;(*modus*)
		faktor :	UDINT;(*Systemtakt-Faktor*)
		init :	BOOL;
		v_plc_ticks_per_sec :	UDINT;
		base :	UDINT := UDINT#1000;
	END_VAR

	IF init = FALSE THEN
		v_plc_ticks_per_sec := INT_TO_UDINT(PLC_TICKS_PER_SEC);
		IF v_plc_ticks_per_sec = UDINT#1024 THEN
			faktor := UDINT#1;
			mode := FALSE;
		ELSIF v_plc_ticks_per_sec > UDINT#0 THEN
			IF v_plc_ticks_per_sec <= base THEN
				faktor := base / v_plc_ticks_per_sec;
				mode := FALSE;
			ELSE
				faktor := v_plc_ticks_per_sec / base;
				mode := TRUE;
			END_IF;
		ELSE
			faktor := UDINT#1;
		END_IF;
		init := TRUE;
	END_IF;

	IF mode THEN
		IF mode THEN
		    T_PLC_MS := DINT_TO_UDINT(PLC_SYS_TICK_CNT) * faktor;
		ELSE
		    T_PLC_MS := DINT_TO_UDINT(PLC_SYS_TICK_CNT) / faktor;
		END_IF;
	ELSE
		T_PLC_MS := DINT_TO_UDINT(PLC_SYS_TICK_CNT) * faktor;
	END_IF;

	IF debug THEN
		T_PLC_MS := (DWORD_TO_UDINT(SHL(UDINT_TO_DWORD(T_PLC_MS),N) OR SHL(temp,N)) - UDINT#1) + Offset;
	END_IF;

END_FUNCTION_BLOCK

FUNCTION_BLOCK CLK_PRG
	VAR_INPUT
		PT :	TIME := T#10ms;
	END_VAR

	VAR_OUTPUT
		Q :	BOOL;
	END_VAR

	VAR
		init :	BOOL := FALSE;
		last :	TIME;
		tx :	TIME;
		T_PLC_MS :	T_PLC_MS_block;
	END_VAR

	T_PLC_MS();
	tx:= UDINT_TO_TIME(T_PLC_MS.T_PLC_MS);

	IF NOT init THEN
		init := TRUE;
		last := tx - pt;
	END_IF;

	Q := tx - last >= pt;
	IF Q THEN last := tx; END_IF;
END_FUNCTION_BLOCK

FUNCTION _REAL_TO_UDINT:UDINT
  VAR_INPUT
    X :	REAL;
  END_VAR

  IF REAL_TO_UDINT(0.5) = UDINT#1 THEN
    _REAL_TO_UDINT := REAL_TO_UDINT(x);
  ELSIF X > 0.0 THEN
    _REAL_TO_UDINT := REAL_TO_UDINT(x+0.5);
  ELSIF X < 0.0 THEN
    _REAL_TO_UDINT := REAL_TO_UDINT(x-0.5);
  ELSE
    _REAL_TO_UDINT := UDINT#0;
  END_IF;
END_FUNCTION

FUNCTION REAL_TO_TIME2:TIME
	VAR_INPUT
		IN :	REAL;
	END_VAR

	REAL_TO_TIME2 := DINT_TO_TIME(UDINT_TO_DINT(_REAL_TO_UDINT(IN)));
END_FUNCTION

FUNCTION_BLOCK TP_X
	VAR_INPUT
		IN :	BOOL;
		PT :	TIME;
	END_VAR

	VAR_OUTPUT
		Q :	BOOL;
		ET :	TIME;
	END_VAR

	VAR
		edge :	BOOL;
		start :	TIME;
		tx :	TIME;
		T_PLC_MS :	T_PLC_MS_block;
	END_VAR

	T_PLC_MS();
	tx := UDINT_TO_TIME(T_PLC_MS.T_PLC_MS);

	IF IN AND NOT edge THEN
		start := tx;
		Q := PT > t#0ms;
	ELSIF Q THEN
		ET := tx - start;
		IF ET >= PT THEN
			Q := FALSE;
			ET := t#0ms;
		END_IF;
	END_IF;
	edge := IN;

END_FUNCTION_BLOCK

FUNCTION_BLOCK PWM_DC
	VAR_INPUT
		F :	REAL;
		DC :	REAL;
	END_VAR

	VAR_OUTPUT
		Q :	BOOL;
	END_VAR

	VAR
		clk :	CLK_Prg;
		pulse :	TP_X;
		tmp :	REAL;
	END_VAR

	IF F > 0.0 THEN
		tmp := 1000.0/F;
		CLK(PT := REAL_TO_TIME2(tmp));
		Pulse(in := clk.Q, pt := REAL_TO_TIME2(tmp*DC));
		Q := pulse.Q;
	END_IF;
END_FUNCTION_BLOCK

FUNCTION_BLOCK CTRL_PWM
	VAR_INPUT
		CI :	REAL;
		MAN_IN :	REAL;
		MANUAL :	BOOL;
		F :	REAL;
	END_VAR

	VAR_OUTPUT
		Q :	BOOL;
	END_VAR

	VAR
		PW :	PWM_DC;
	END_VAR

	PW(F := F, DC := SEL(MANUAL,CI,MAN_IN));
	Q := PW.Q;
END_FUNCTION_BLOCK

PROGRAM program0
  VAR
	CI     :	REAL;
	MAN_IN :	REAL;
	MANUAL :	BOOL;
	F      :	REAL;

	Q :	BOOL;

	func_block : CTRL_PWM;
  END_VAR
	func_block.CI    :=CI    ;
	func_block.MAN_IN:=MAN_IN;
	func_block.MANUAL:=MANUAL;
	func_block.F     :=F     ;
	func_block();
	Q := func_block.Q;
END_PROGRAM

CONFIGURATION Config0
	VAR_GLOBAL
		PLC_TICKS_PER_SEC :	INT;
		PLC_SYS_TICK_CNT :	DINT;
	END_VAR

  RESOURCE Res0 ON PLC
    TASK task0(INTERVAL := T#20ms,PRIORITY := 0);
    PROGRAM instance0 WITH task0 : program0;
  END_RESOURCE
END_CONFIGURATION

(* ---- lb_claude_assisted_8f41420342e6_0017.st ---- *)
FUNCTION_BLOCK SW_RECONFIG_Block

	VAR_INPUT
		IN :	BOOL;
		TD :	TIME;
		TR :	TIME;
	END_VAR

	VAR_OUTPUT
		Q :	BOOL;
	END_VAR

	VAR
		T1 :	TON;
		T2 :	TON;
		INV :	BOOL;
	END_VAR

	t1(in := IN, PT := TD);

	IF tr > t#0s THEN
		Q := t1.Q XOR inv;
		T2(in := Q, pt := TR);
		IF T2.Q THEN INV := NOT INV; END_IF;
	ELSE
		Q := t1.Q;
	END_IF;

END_FUNCTION_BLOCK

FUNCTION_BLOCK CLICK_MODE_Block

	VAR_INPUT
		IN :	BOOL;
		T_LONG :	TIME := T#500ms;
	END_VAR

	VAR_OUTPUT
		SINGLE :	BOOL;
		DOUBLE :	BOOL;
		LONG :	BOOL;
		TP_LONG :	BOOL;
	END_VAR

	VAR
		Timer :	TP;
		cnt :	INT;
		last :	BOOL;
	END_VAR

	timer(in := IN, PT := T_LONG);
	single := FALSE;
	double := FALSE;

	IF timer.Q THEN
		IF NOT in AND last THEN	cnt := cnt + 1; END_IF;
	ELSE
		CASE cnt OF
			1 : single := TRUE;
			2 : double := TRUE;
		END_CASE;
		cnt := 0;
	END_IF;
	last := in;
	TP_LONG := NOT timer.Q AND (NOT LONG) AND IN;
	LONG := NOT timer.Q AND in;

END_FUNCTION_BLOCK

FUNCTION UDINT_TO_TIME2:TIME

	VAR_INPUT
		IN :	UDINT;
	END_VAR

	UDINT_TO_TIME2 := DINT_TO_TIME(UDINT_TO_DINT(IN));

END_FUNCTION

FUNCTION_BLOCK T_PLC_MS_block
	VAR_OUTPUT
		T_PLC_MS :	UDINT;
	END_VAR

	VAR_EXTERNAL
		PLC_TICKS_PER_SEC :	INT;
		PLC_SYS_TICK_CNT :	DINT;
	END_VAR

	VAR
		debug :	BOOL;(*Debug-Mode ON / OFF*)
		N :	INT;(*Debug-Faktor*)
		Offset :	UDINT;(*Debug-Offset*)
		temp :	DWORD := DWORD#1;(*Debug-Offset*)
		mode :	BOOL;(*modus*)
		faktor :	UDINT;(*Systemtakt-Faktor*)
		init :	BOOL;
		v_plc_ticks_per_sec :	UDINT;
		base :	UDINT := UDINT#1000;
	END_VAR

	IF init = FALSE THEN
		v_plc_ticks_per_sec := INT_TO_UDINT(PLC_TICKS_PER_SEC);
		IF v_plc_ticks_per_sec = UDINT#1024 THEN
			faktor := UDINT#1;
			mode := FALSE;
		ELSIF v_plc_ticks_per_sec > UDINT#0 THEN
			IF v_plc_ticks_per_sec <= base THEN
				faktor := base / v_plc_ticks_per_sec;
				mode := FALSE;
			ELSE
				faktor := v_plc_ticks_per_sec / base;
				mode := TRUE;
			END_IF;
		ELSE
			faktor := UDINT#1;
		END_IF;
		init := TRUE;
	END_IF;

	IF mode THEN
		T_PLC_MS := DINT_TO_UDINT(PLC_SYS_TICK_CNT) / faktor;
	ELSE
		T_PLC_MS := DINT_TO_UDINT(PLC_SYS_TICK_CNT) * faktor;
	END_IF;

	IF debug THEN
		T_PLC_MS := (DWORD_TO_UDINT(SHL(UDINT_TO_DWORD(T_PLC_MS),N) OR SHL(temp,N)) - UDINT#1) + Offset;
	END_IF;

END_FUNCTION_BLOCK

FUNCTION TIME_TO_UDINT2:UDINT
	VAR_INPUT
		X :	TIME;
	END_VAR

	TIME_TO_UDINT2 := DINT_TO_UDINT(TIME_TO_DINT(X));
END_FUNCTION

FUNCTION FRMP_B:BYTE
	VAR_INPUT
		START :	BYTE;
		DIR :	BOOL;
		TD :	TIME;
		TR :	TIME;
	END_VAR

	IF TD < TR THEN
		FRMP_B := MIN(UDINT_TO_BYTE(DWORD_TO_UDINT(SHL(TIME_TO_DWORD(TD), 8)) / TIME_TO_UDINT2(TR)), SEL(DIR, START, USINT_TO_BYTE(USINT#255 - BYTE_TO_USINT(START))));
		IF DIR THEN
			FRMP_B := USINT_TO_BYTE(BYTE_TO_USINT(START) + BYTE_TO_USINT(FRMP_B));
		ELSE
			FRMP_B := USINT_TO_BYTE(BYTE_TO_USINT(START) - BYTE_TO_USINT(FRMP_B));
		END_IF;
	ELSE
		FRMP_B := SEL(DIR, BYTE#0, BYTE#255);
	END_IF;
END_FUNCTION

FUNCTION_BLOCK _RMP_B
	VAR_INPUT
		DIR :	BOOL;
		E :	BOOL := TRUE;
		TR :	TIME;
	END_VAR

	VAR_IN_OUT
		RMP :	BYTE;
	END_VAR

	VAR
		T_PLC_MS :	T_PLC_MS_block;
		tx :	TIME;
		tl :	TIME;
		tn :	TIME;
		init :	BOOL;
		last_dir :	BOOL;
		start :	BYTE;
	END_VAR

	T_PLC_MS();
	tx := UDINT_TO_TIME(T_PLC_MS.T_PLC_MS);

	IF E AND init AND (dir = last_dir) AND (RMP <> SEL(DIR, BYTE#0, BYTE#255)) AND TR = tn THEN
		RMP := FRMP_B(start, DIR, tx - tl, TR);
	ELSE
		init := TRUE;
		tl := tx;
		tn := tr;
		start := RMP;
	END_IF;
	last_dir := dir;
END_FUNCTION_BLOCK

FUNCTION _BYTE_TO_INT:INT
	VAR_INPUT
		IN :	BYTE;
	END_VAR

	_BYTE_TO_INT := USINT_TO_INT(BYTE_TO_USINT(IN));
END_FUNCTION

FUNCTION_BLOCK DIMM_I_Block

	VAR_INPUT
		SET :	BOOL;
		VAL :	BYTE := BYTE#255;
		IN :	BOOL;
		RST :	BOOL;
		T_DEBOUNCE :	TIME := T#10ms;
		T_RECONFIG :	TIME := T#10s;
		T_ON_MAX :	TIME := T#0h;
		T_DIMM_START :	TIME := T#1s;
		T_DIMM :	TIME := T#3s;
		MIN_ON :	BYTE := BYTE#50;
		MAX_ON :	BYTE := BYTE#255;
		SOFT_DIMM :	BOOL := TRUE;
		DBL_TOGGLE :	BOOL;
		RST_OUT :	BOOL;
	END_VAR

	VAR_OUTPUT
		Q :	BOOL;
		DBL :	BOOL;
	END_VAR

	VAR_IN_OUT
		OUT :	BYTE;
	END_VAR

	VAR
		config :	SW_RECONFIG_Block;
		decode :	CLICK_MODE_Block;
		t3 :	TON;
		dim :	_RMP_B;
		dir :	BOOL;
	END_VAR

	config(IN := IN, TD := T_DEBOUNCE, TR := T_RECONFIG);
	decode(in := config.Q, T_LONG := T_DIMM_START);

	IF RST THEN
		IF rst_out THEN out := BYTE#0; END_IF;
		Q := FALSE;
		dir := out > BYTE#127;
	ELSIF set THEN
		out := val;
		Q := TRUE;
		dir := out > BYTE#127;
	ELSIF decode.SINGLE THEN
		Q := NOT Q;
		IF Q THEN OUT := INT_TO_BYTE(LIMIT_INT(MAX(_BYTE_TO_INT(MIN_ON),1), _BYTE_TO_INT(out), _BYTE_TO_INT(MAX_ON)));	END_IF;
		dir := OUT > BYTE#127;
	ELSIF decode.TP_LONG THEN
		IF NOT Q THEN
			IF SOFT_DIMM THEN
				OUT := BYTE#1;
				dir := TRUE;
			ELSE
				out := INT_TO_BYTE(LIMIT_INT(MAX(_BYTE_TO_INT(MIN_ON),1), _BYTE_TO_INT(out), _BYTE_TO_INT(MAX_ON)));
				DIR := out < BYTE#127;
			END_IF;
			Q := TRUE;
		ELSE
			dir := NOT dir;
		END_IF;
	END_IF;

	IF NOT dbl_toggle THEN dbl := FALSE; END_IF;
	IF decode.DOUBLE THEN dbl := NOT dbl; END_IF;

	dim(DIR := dir, e := decode.LONG AND Q, TR := T_DIMM, rmp := out);
	OUT := dim.RMP;
	IF out = BYTE#0 THEN
		dir := TRUE;
	ELSIF out = BYTE#255 THEN
		dir := FALSE;
	END_IF;

	IF t_ON_MAX > t#0s THEN
		IF t_ON_MAX > t#0s THEN
		    t3(in := q, PT := T#9999h);
		ELSE
		    t3(in := q, pt := T_ON_MAX);
		END_IF;
		Q := Q XOR t3.Q;
	END_IF;

END_FUNCTION_BLOCK

PROGRAM program0
	VAR
	    SET :	BOOL;
		VAL :	BYTE := BYTE#255;
		IN :	BOOL;
		RST :	BOOL;
		T_DEBOUNCE :	TIME := T#10ms;
		T_RECONFIG :	TIME := T#10s;
		T_ON_MAX :	TIME := T#0h;
		T_DIMM_START :	TIME := T#1s;
		T_DIMM :	TIME := T#3s;
		MIN_ON :	BYTE := BYTE#50;
		MAX_ON :	BYTE := BYTE#255;
		SOFT_DIMM :	BOOL := TRUE;
		DBL_TOGGLE :	BOOL;
		RST_OUT :	BOOL;
		OUT :	BYTE;
		Q :	BOOL;
		DBL :	BOOL;

		func_block : DIMM_I_Block;
  	END_VAR
	func_block.SET := SET;
	func_block.VAL := VAL;
	func_block.IN := IN;
	func_block.RST := RST;
	func_block.T_DEBOUNCE := T_DEBOUNCE;
	func_block.T_RECONFIG := T_RECONFIG;
	func_block.T_ON_MAX := T_ON_MAX;
	func_block.T_DIMM_START := T_DIMM_START;
	func_block.T_DIMM := T_DIMM;
	func_block.MIN_ON := MIN_ON;
	func_block.MAX_ON := MAX_ON;
	func_block.SOFT_DIMM := SOFT_DIMM;
	func_block.DBL_TOGGLE := DBL_TOGGLE;
	func_block.RST_OUT := RST_OUT;
	func_block.OUT := OUT;

	func_block();
	OUT := func_block.OUT;
	Q := func_block.Q;
	DBL := func_block.DBL;
END_PROGRAM

CONFIGURATION Config0
	VAR_GLOBAL
		PLC_TICKS_PER_SEC :	INT;
		PLC_SYS_TICK_CNT :	DINT;
	END_VAR
  	RESOURCE Res0 ON PLC
    	TASK task0(INTERVAL := T#20ms,PRIORITY := 0);
    	PROGRAM instance0 WITH task0 : program0;
  	END_RESOURCE
END_CONFIGURATION

(* ---- lb_claude_assisted_936342dc23ae_0088.st ---- *)
TYPE
  LOGLEVEL : (CRITICAL, WARNING, INFO, DEBUG) := INFO;
END_TYPE

FUNCTION_BLOCK LOGGER
  VAR_INPUT
    TRIG : BOOL;
    MSG : STRING;
    LEVEL : LOGLEVEL := INFO;
  END_VAR
  VAR
    TRIG0 : BOOL;
  END_VAR

  IF TRIG AND NOT TRIG0 THEN
  {{
   LogMessage(GetFbVar(LEVEL),(char*)GetFbVar(MSG, .body),GetFbVar(MSG, .len));
  }}
  END_IF;
  TRIG0:=TRIG;
END_FUNCTION_BLOCK

FUNCTION_BLOCK python_eval
  VAR_INPUT
    TRIG : BOOL;
    CODE : STRING;
  END_VAR
  VAR_OUTPUT
    ACK : BOOL;
    RESULT : STRING;
  END_VAR
  VAR
    STATE : DWORD;
    BUFFER : STRING;
    PREBUFFER : STRING;
    TRIGM1 : BOOL;
    TRIGGED : BOOL;
  END_VAR

  {extern void __PythonEvalFB(int, PYTHON_EVAL*);__PythonEvalFB(0, data__);}
END_FUNCTION_BLOCK

FUNCTION_BLOCK python_poll
  VAR_INPUT
    TRIG : BOOL;
    CODE : STRING;
  END_VAR
  VAR_OUTPUT
    ACK : BOOL;
    RESULT : STRING;
  END_VAR
  VAR
    STATE : DWORD;
    BUFFER : STRING;
    PREBUFFER : STRING;
    TRIGM1 : BOOL;
    TRIGGED : BOOL;
  END_VAR

  {extern void __PythonEvalFB(int, PYTHON_EVAL*);__PythonEvalFB(1,(PYTHON_EVAL*)(void*)data__);}
END_FUNCTION_BLOCK

FUNCTION_BLOCK python_gear
  VAR_INPUT
    N : UINT;
    TRIG : BOOL;
    CODE : STRING;
  END_VAR
  VAR_OUTPUT
    ACK : BOOL;
    RESULT : STRING;
  END_VAR
  VAR
    py_eval : python_eval;
    COUNTER : UINT;
    ADD10_OUT : UINT;
    EQ13_OUT : BOOL;
    SEL15_OUT : UINT;
    AND7_OUT : BOOL;
  END_VAR

  ADD10_OUT := ADD(COUNTER, 1);
  EQ13_OUT := EQ(N, ADD10_OUT);
  SEL15_OUT := SEL(EQ13_OUT, ADD10_OUT, 0);
  COUNTER := SEL15_OUT;
  AND7_OUT := AND(EQ13_OUT, TRIG);
  py_eval(TRIG := AND7_OUT, CODE := CODE);
  ACK := py_eval.ACK;
  RESULT := py_eval.RESULT;
END_FUNCTION_BLOCK

PROGRAM Gate_Controller
  VAR
    Start_Loop : BOOL := False;
    one_hour : TIME := T#1h;
    One_Hour_Timer : TON;
    Gate_Open : BOOL := False;
  END_VAR
  VAR_OUTPUT
    Close_Gate_Inst : BOOL := False;
  END_VAR
  VAR_INPUT
    Sensed_Car : BOOL := False;
    Sensed_Car_Inst : BOOL := False;
    Sensed_App : BOOL := False;
    Mobile_Inst : BOOL := False;
    Mobile_Auth : STRING;
  END_VAR
  VAR
    my_defined_str : STRING := '"1234"';
  END_VAR

  One_Hour_Timer(IN := NOT(Start_Loop), PT := one_hour);

  IF One_Hour_Timer.Q THEN
    IF Gate_Open THEN
      Close_Gate_Inst := True;
      Gate_Open := False;
    END_IF;
  END_IF;

  IF Sensed_App THEN
    (* How can I do some authentication here? *)
    IF EQ(Mobile_Auth, my_defined_str) THEN
      Close_Gate_Inst := XOR(Mobile_Inst, Gate_Open);
      IF EQ(Mobile_Auth, my_defined_str) THEN
          Gate_Open := False;
      ELSE
          Gate_Open := Mobile_Inst;
      END_IF;
    END_IF;
  END_IF;

  IF AND(Sensed_Car, Sensed_Car_Inst) THEN
    Close_Gate_Inst := XOR(Sensed_Car_Inst, Gate_Open);
    Gate_Open := Sensed_Car_Inst;
  END_IF;

  Start_Loop := One_Hour_Timer.Q;
END_PROGRAM

CONFIGURATION Config0

  RESOURCE Res0 ON PLC
    TASK task0(INTERVAL := T#20ms,PRIORITY := 0);
    PROGRAM instance0 WITH task0 : Gate_Controller;
  END_RESOURCE
END_CONFIGURATION

(* ---- lb_claude_assisted_937718607de8_0124.st ---- *)
FUNCTION BIT_LOAD_B:BYTE
	VAR_INPUT
		IN :	BYTE;
		VAL :	BOOL;
		POS :	INT;
	END_VAR

	IF VAL THEN
		BIT_LOAD_B := in OR SHL(BYTE#1,pos);
	ELSE
		BIT_LOAD_B := in AND (NOT SHL(BYTE#1,pos));
	END_IF;
END_FUNCTION

FUNCTION_BLOCK INTERLOCK_4_Block

	VAR_INPUT
		I0 :	BOOL;
		I1 :	BOOL;
		I2 :	BOOL;
		I3 :	BOOL;
		E :	BOOL;
		MODE :	INT;
	END_VAR

	VAR_OUTPUT
		OUT :	BYTE;
		_TP :	BOOL;
	END_VAR

	VAR
		in :	BYTE;
		last :	BYTE;
		old :	BYTE;
		lmode :	INT;
	END_VAR

	IF E THEN
	(* reset all vars when there is a mode change on thy fly *)
		IF mode <> lmode THEN
			out := BYTE#0;
			last := BYTE#0;
			old := BYTE#0;
			IF mode <> lmode THEN
			    lmode := 0;
			ELSE
			    lmode := mode;
			END_IF;
		END_IF;
		(* load inputs into in *)
		in:=BIT_LOAD_B(in,I0,0); (* in.0 *)
		in:=BIT_LOAD_B(in,I1,1); (* in.1 *)
		in:=BIT_LOAD_B(in,I2,2); (* in.2 *)
		in:=BIT_LOAD_B(in,I3,3); (* in.3 *)
		(* only execute when there is any change *)
		IF in <> last THEN
			(* only execute when inputs have chages state *)
			CASE mode OF
				0:	(* output directly display inputs as bits in byte out *)
					out := in;

				1:	(* the input with the highest number will be acepted *)
					IF    (in AND BYTE#2#00001000) > BYTE#0 (* in.3 *) THEN out := BYTE#8;
					ELSIF (in AND BYTE#2#00000100) > BYTE#0 (* in.2 *) THEN out := BYTE#4;
					ELSIF (in AND BYTE#2#00000010) > BYTE#0 (* in.1 *) THEN out := BYTE#2;
					ELSE out := in;
					END_IF;

				2:	(* input last pressed will be displayed only *)
					last := ((in XOR last) AND in);
					IF    (last AND BYTE#2#00001000) > BYTE#0 (* last.3 *) THEN out := BYTE#8;
					ELSIF (last AND BYTE#2#00000100) > BYTE#0 (* last.2 *) THEN out := BYTE#4;
					ELSIF (last AND BYTE#2#00000010) > BYTE#0 (* last.1 *) THEN out := BYTE#2;
					ELSE out := last;
					END_IF;

				3:	(* any input active will disable all other inputs *)
					IF (out AND in) = BYTE#0 THEN
						IF    (in AND BYTE#2#00001000) > BYTE#0 (* in.3 *) THEN out := BYTE#8;
						ELSIF (in AND BYTE#2#00000100) > BYTE#0 (* in.2 *) THEN out := BYTE#4;
						ELSIF (in AND BYTE#2#00000010) > BYTE#0 (* in.1 *) THEN out := BYTE#2;
						ELSE out := in;
						END_IF;
					END_IF;

			END_CASE;
			last := in;
		END_IF;
		_tp := out <> old;
		old := out;
	ELSE
		out := BYTE#0;
		last := BYTE#0;
		old := BYTE#0;
		lmode := 0;
		_tp := FALSE;
	END_IF;

END_FUNCTION_BLOCK

PROGRAM program0

	VAR
		I0 :	BOOL;
		I1 :	BOOL;
		I2 :	BOOL;
		I3 :	BOOL;
		E :	BOOL;
		MODE :	INT;
		OUT :	BYTE;
		_TP :	BOOL;
		func_block : INTERLOCK_4_Block;
	END_VAR
	func_block.I0 := I0;
	func_block.I1 := I1;
	func_block.I2 := I2;
	func_block.I3 := I3;
	func_block.E := E;
	func_block.MODE := MODE;
	func_block();
	OUT := func_block.OUT;
	_TP := func_block._TP;

END_PROGRAM

CONFIGURATION Config0

	RESOURCE Res0 ON PLC
		TASK task0(INTERVAL := T#20ms,PRIORITY := 0);
		PROGRAM instance0 WITH task0 : program0;
	END_RESOURCE

END_CONFIGURATION

(* ---- lb_claude_assisted_9410414c6070_0036.st ---- *)
FUNCTION_BLOCK T_PLC_MS_block
	VAR_OUTPUT
		T_PLC_MS :	UDINT;
	END_VAR

	VAR_EXTERNAL
		PLC_TICKS_PER_SEC :	INT;
		PLC_SYS_TICK_CNT :	DINT;
	END_VAR

	VAR
		debug :	BOOL;(*Debug-Mode ON / OFF*)
		N :	INT;(*Debug-Faktor*)
		Offset :	UDINT;(*Debug-Offset*)
		temp :	DWORD := DWORD#1;(*Debug-Offset*)
		mode :	BOOL;(*modus*)
		faktor :	UDINT;(*Systemtakt-Faktor*)
		init :	BOOL;
		v_plc_ticks_per_sec :	UDINT;
		base :	UDINT := UDINT#1000;
	END_VAR

	IF init = FALSE THEN
		v_plc_ticks_per_sec := INT_TO_UDINT(PLC_TICKS_PER_SEC);
		IF v_plc_ticks_per_sec = UDINT#1024 THEN
			faktor := UDINT#1;
			mode := FALSE;
		ELSIF v_plc_ticks_per_sec > UDINT#0 THEN
			IF v_plc_ticks_per_sec <= base THEN
				faktor := base / v_plc_ticks_per_sec;
				mode := FALSE;
			ELSE
				faktor := v_plc_ticks_per_sec / base;
				mode := TRUE;
			END_IF;
		ELSE
			faktor := UDINT#1;
		END_IF;
		init := TRUE;
	END_IF;

	IF mode THEN
		T_PLC_MS := DINT_TO_UDINT(PLC_SYS_TICK_CNT) / faktor;
	ELSE
		T_PLC_MS := DINT_TO_UDINT(PLC_SYS_TICK_CNT) * faktor;
	END_IF;

	IF debug THEN
		T_PLC_MS := (DWORD_TO_UDINT(SHL(UDINT_TO_DWORD(T_PLC_MS),N) OR SHL(temp,N)) - UDINT#1) + Offset;
	END_IF;
END_FUNCTION_BLOCK

FUNCTION_BLOCK FT_PROFILE

	VAR_INPUT
		K :	REAL := 1.0;
		O :	REAL := 0.0;
		M :	REAL := 1.0;
		E :	BOOL;
		VALUE_0 :	REAL;
		TIME_1 :	TIME;
		VALUE_1 :	REAL;
		TIME_2 :	TIME;
		VALUE_2 :	REAL;
		TIME_3 :	TIME;
		VALUE_3 :	REAL;
		TIME_10 :	TIME;
		VALUE_10 :	REAL;
		TIME_11 :	TIME;
		VALUE_11 :	REAL;
		TIME_12 :	TIME;
		VALUE_12 :	REAL;
		TIME_13 :	TIME;
		VALUE_13 :	REAL;
	END_VAR

	VAR_OUTPUT
		Y :	REAL;
		RUN :	BOOL;
		ET :	TIME;
	END_VAR

	VAR
		tx :	TIME;
		edge :	BOOL;
		state :	INT;
		ta :	TIME;
		tb :	TIME;
		t0 :	TIME;
		temp :	REAL;
		va :	REAL;
		vb :	REAL;
		T_PLC_MS :	T_PLC_MS_block;
	END_VAR

	T_PLC_MS();
	tx:= UDINT_TO_TIME(T_PLC_MS.T_PLC_MS);

	(* determine start condition *)
	IF E AND NOT edge THEN
		RUN := TRUE;
		ET := t#0s;
		t0 := tx;
		ta := tx;
		tb := multime(time_1, M);
		va := value_0;
		vb := value_1;
		temp := value_0;
		state := 1;
	END_IF;
	edge := E;

	(* generate startup profile *)
	IF run THEN
		CASE state OF
			1:	IF tx - ta >= tb THEN
					ta := ta + tb;
					tb := multime(time_2 - time_1, M);
					va := value_1;
					vb := value_2;
					temp := value_1;
					IF tx - ta >= tb THEN
					    state := 1;
					ELSE
					    state := 2;
					END_IF;
				ELSE
					temp := ((vb - va) * TIME_TO_REAL(tx - ta) / TIME_TO_REAL(tb) + va);
				END_IF;
			2:	IF tx - ta >= tb THEN
					ta := ta + tb;
					tb := multime(time_3 - time_2, M);
					va := value_2;
					vb := value_3;
					temp := value_2;
					state := 3;
				ELSE
					temp := ((vb - va) * TIME_TO_REAL(tx - ta) / TIME_TO_REAL(tb) + va);
				END_IF;
			3:	IF tx - ta >= tb THEN
					ta := ta + tb;
					tb := multime(time_10 - time_3, M);
					va := value_3;
					vb := value_10;
					temp := value_3;
					state := 4;
				ELSE
					temp := ((vb - va) * TIME_TO_REAL(tx - ta) / TIME_TO_REAL(tb) + va);
				END_IF;
			4 :	IF tx - ta >= tb THEN
					ta := ta + tb;
					tb := multime(time_11 - time_10, M);
					va := value_10;
					vb := value_11;
					temp := value_10;
					IF E THEN state := 5; ELSE state := 6; END_IF;
				ELSE
					temp := ((vb - va) * TIME_TO_REAL(tx - ta) / TIME_TO_REAL(tb) + va);
				END_IF;
			5:	(* extend the signal while E is true *)
				IF E THEN
					ta := tx;
				ELSE
					state := 6;
				END_IF;
			6:	IF tx - ta >= tb THEN
					ta := ta + tb;
					tb := multime(time_12 - time_11, M);
					va := value_11;
					vb := value_12;
					temp := value_11;
					state := 7;
				ELSE
					temp := ((vb - va) * TIME_TO_REAL(tx - ta) / TIME_TO_REAL(tb) + va);
				END_IF;
			7:	IF tx - ta >= tb THEN
					ta := ta + tb;
					tb := multime(time_13 - time_12, M);
					va := value_12;
					vb := value_13;
					temp := value_12;
					state := 8;
				ELSE
					temp := ((vb - va) * TIME_TO_REAL(tx - ta) / TIME_TO_REAL(tb) + va);
				END_IF;
			8:	IF tx - ta >= tb THEN
					temp := value_13;
					run := FALSE;
				ELSE
					temp := ((vb - va) * TIME_TO_REAL(tx - ta) / TIME_TO_REAL(tb) + va);
				END_IF;
		END_CASE;
		Y := temp * K + O;
		ET := tx - t0;
	END_IF;

END_FUNCTION_BLOCK

PROGRAM program0
	VAR
		K :	REAL := 1.0;
		O :	REAL := 0.0;
		M :	REAL := 1.0;
		E :	BOOL;
		VALUE_0 :	REAL;
		TIME_1 :	TIME;
		VALUE_1 :	REAL;
		TIME_2 :	TIME;
		VALUE_2 :	REAL;
		TIME_3 :	TIME;
		VALUE_3 :	REAL;
		TIME_10 :	TIME;
		VALUE_10 :	REAL;
		TIME_11 :	TIME;
		VALUE_11 :	REAL;
		TIME_12 :	TIME;
		VALUE_12 :	REAL;
		TIME_13 :	TIME;
		VALUE_13 :	REAL;

		Y :	REAL;
		RUN :	BOOL;
		ET :	TIME;

		func_block : FT_PROFILE;
	END_VAR
	func_block.K  := K ;
	func_block.O  := O ;
	func_block.M  := M ;
	func_block.E  := E ;
	func_block.VALUE_0  := VALUE_0 ;
	func_block.TIME_1  := TIME_1 ;
	func_block.VALUE_1  := VALUE_1 ;
	func_block.TIME_2  := TIME_2 ;
	func_block.VALUE_2  := VALUE_2 ;
	func_block.TIME_3  := TIME_3 ;
	func_block.VALUE_3  := VALUE_3 ;
	func_block.TIME_10  := TIME_10 ;
	func_block.VALUE_10  := VALUE_10 ;
	func_block.TIME_11  := TIME_11 ;
	func_block.VALUE_11  := VALUE_11 ;
	func_block.TIME_12  := TIME_12 ;
	func_block.VALUE_12  := VALUE_12 ;
	func_block.TIME_13  := TIME_13 ;
	func_block.VALUE_13  := VALUE_13 ;
	func_block();
	Y := func_block.Y;
	RUN := func_block.RUN;
	ET := func_block.ET;
END_PROGRAM

CONFIGURATION Config0

	VAR_GLOBAL
		PLC_TICKS_PER_SEC :	INT;
		PLC_SYS_TICK_CNT :	DINT;
	END_VAR

	RESOURCE Res0 ON PLC
		TASK task0(INTERVAL := T#20ms,PRIORITY := 0);
		PROGRAM instance0 WITH task0 : program0;
	END_RESOURCE

END_CONFIGURATION

(* ---- lb_claude_assisted_951ec4f842da_0009.st ---- *)
FUNCTION_BLOCK T_PLC_MS_block
	VAR_OUTPUT
		T_PLC_MS :	UDINT;
	END_VAR

	VAR_EXTERNAL
		PLC_TICKS_PER_SEC :	INT;
		PLC_SYS_TICK_CNT :	DINT;
	END_VAR

	VAR
		debug :	BOOL;(*Debug-Mode ON / OFF*)
		N :	INT;(*Debug-Faktor*)
		Offset :	UDINT;(*Debug-Offset*)
		temp :	DWORD := DWORD#1;(*Debug-Offset*)
		mode :	BOOL;(*modus*)
		faktor :	UDINT;(*Systemtakt-Faktor*)
		init :	BOOL;
		v_plc_ticks_per_sec :	UDINT;
		base :	UDINT := UDINT#1000;
	END_VAR

	IF init = FALSE THEN
		v_plc_ticks_per_sec := INT_TO_UDINT(PLC_TICKS_PER_SEC);
		IF v_plc_ticks_per_sec = UDINT#1024 THEN
			faktor := UDINT#1;
			mode := FALSE;
		ELSIF v_plc_ticks_per_sec > UDINT#0 THEN
			IF v_plc_ticks_per_sec <= base THEN
				faktor := base / v_plc_ticks_per_sec;
				mode := FALSE;
			ELSE
				faktor := v_plc_ticks_per_sec / base;
				mode := TRUE;
			END_IF;
		ELSE
			faktor := UDINT#1;
		END_IF;
		init := TRUE;
	END_IF;

	IF mode THEN
		T_PLC_MS := DINT_TO_UDINT(PLC_SYS_TICK_CNT) / faktor;
	ELSE
		IF NOT mode THEN
		    T_PLC_MS := DINT_TO_UDINT(PLC_SYS_TICK_CNT) / faktor;
		ELSE
		    T_PLC_MS := DINT_TO_UDINT(PLC_SYS_TICK_CNT) * faktor;
		END_IF;
	END_IF;

	IF debug THEN
		T_PLC_MS := (DWORD_TO_UDINT(SHL(UDINT_TO_DWORD(T_PLC_MS),N) OR SHL(temp,N)) - UDINT#1) + Offset;
	END_IF;
END_FUNCTION_BLOCK

FUNCTION_BLOCK INTEGRATE

	VAR_INPUT
		E :	BOOL := TRUE;
		X :	REAL;
		K :	REAL := 1.0;
	END_VAR

	VAR_IN_OUT
		Y :	REAL;
	END_VAR

	VAR
		X_last :	REAL;
		init :	BOOL;
		T_PLC_MS :	T_PLC_MS_block;
		last :	UDINT;
		tx :	UDINT;
	END_VAR

	T_PLC_MS();
	tx:= T_PLC_MS.T_PLC_MS;

	IF NOT init THEN
		init := TRUE;
		X_last := X;
	ELSIF E THEN
		Y := (X + X_LAST) * 0.5E-3 * UDINT_TO_REAL(tx-last) * K + Y;
		X_last := X;
	END_IF;
	last := tx;

END_FUNCTION_BLOCK

FUNCTION_BLOCK FT_PT2

	VAR_INPUT
		IN :	REAL;
		T :	TIME;
		D :	REAL;
		K :	REAL := 1.0;
	END_VAR

	VAR_OUTPUT
		OUT :	REAL;
	END_VAR

	VAR
		init :	BOOL;
		int1 :	INTEGRATE;
		int2 :	INTEGRATE;
		tn :	REAL;
		I1 :	REAL;
		I2 :	REAL;
		tn2 :	REAL;
	END_VAR

	IF NOT init OR T = T#0s THEN
		init := TRUE;
		out := K * in;
		I2 := out;
	ELSE
		TN := TIME_TO_REAL(T) / 1000.0;
		tn2 := TN * TN;
		int1(X := in * K / tn2 - I1 * 0.5 * D / TN - I2 / TN2, Y := I1);
		I1 := int1.Y;
		int2(X := I1,Y := I2);
		I2 := int2.Y;
		out := I2;
	END_IF;

END_FUNCTION_BLOCK

PROGRAM program0
	VAR
		IN :	REAL;
		T :	TIME;
		D :	REAL;
		K :	REAL := 1.0;

		OUT :	REAL;

		func_block : FT_PT2;
	END_VAR
	func_block.IN := IN;
	func_block.T := T;
	func_block.D := D;
	func_block.K := K;
	func_block();
	OUT := func_block.OUT;
END_PROGRAM

CONFIGURATION Config0

	VAR_GLOBAL
		PLC_TICKS_PER_SEC :	INT;
		PLC_SYS_TICK_CNT :	DINT;
	END_VAR

	RESOURCE Res0 ON PLC
		TASK task0(INTERVAL := T#20ms,PRIORITY := 0);
		PROGRAM instance0 WITH task0 : program0;
	END_RESOURCE

END_CONFIGURATION

(* ---- lb_claude_assisted_97133923fa41_0098.st ---- *)
FUNCTION_BLOCK GE_0
  VAR_INPUT
    IN1 : DINT;
    IN2 : DINT;
  END_VAR
  VAR_OUTPUT
    OUT : BOOL;
  END_VAR
  VAR
    mytimer : TON;
  END_VAR

  OUT:=FALSE;
  IF IN1>=IN2 then
    OUT:=TRUE;
  END_IF;

  IF mytimer.Q = TRUE THEN
      mytimer(IN := TRUE, PT := T#9999h);
  ELSE
      mytimer(IN := TRUE, PT := t#8000ms);
  END_IF;

  IF mytimer.Q = TRUE then

      OUT:=TRUE;

  End_IF;
END_FUNCTION_BLOCK

PROGRAM PLC3
  VAR_INPUT
    level : DINT;
  END_VAR
  VAR_OUTPUT
    pump : BOOL;
  END_VAR
  VAR
    low : BOOL;
    high : BOOL;
    low_3 : DINT := 0;
    high_3 : DINT := 10;
    GE_00 : GE_0;
    _TMP_LE13_ENO : BOOL;
    _TMP_LE13_OUT : BOOL;
  END_VAR

  GE_00(EN := TRUE, IN1 := level, IN2 := high_3);
  high := GE_00.OUT;
  _TMP_LE13_OUT := LE(EN := TRUE, IN1 := level, IN2 := low_3, ENO => _TMP_LE13_ENO);
  low := _TMP_LE13_OUT;
  pump := NOT(low) AND (high OR pump);
END_PROGRAM

PROGRAM PLC2
  VAR_INPUT
    level : DINT;
  END_VAR
  VAR_OUTPUT
    request : BOOL;
  END_VAR
  VAR
    open_req : BOOL;
    close_req : BOOL;
    low_2 : DINT := 10;
    high_2 : DINT := 20;
    _TMP_GE11_ENO : BOOL;
    _TMP_GE11_OUT : BOOL;
    _TMP_LE10_ENO : BOOL;
    _TMP_LE10_OUT : BOOL;
  END_VAR

  _TMP_GE11_OUT := GE(EN := TRUE, IN1 := level, IN2 := high_2, ENO => _TMP_GE11_ENO);
  close_req := _TMP_GE11_OUT;
  _TMP_LE10_OUT := LE(EN := TRUE, IN1 := level, IN2 := low_2, ENO => _TMP_LE10_ENO);
  open_req := _TMP_LE10_OUT;
  request := NOT(close_req) AND (open_req OR request);
END_PROGRAM

PROGRAM PLC1
  VAR_INPUT
    level : DINT;
    request : DINT;
  END_VAR
  VAR_OUTPUT
    pumps : BOOL;
    valve : BOOL;
  END_VAR
  VAR
    low : BOOL;
    high : BOOL;
    open_req : BOOL;
    close_req : BOOL;
    low_1 : DINT := 40;
    high_1 : DINT := 80;
    _TMP_LE3_ENO : BOOL;
    _TMP_LE3_OUT : BOOL;
    _TMP_GE31_ENO : BOOL;
    _TMP_GE31_OUT : BOOL;
    _TMP_EQ23_ENO : BOOL;
    _TMP_EQ23_OUT : BOOL;
    _TMP_EQ24_ENO : BOOL;
    _TMP_EQ24_OUT : BOOL;
  END_VAR

  _TMP_LE3_OUT := LE(EN := TRUE, IN1 := level, IN2 := low_1, ENO => _TMP_LE3_ENO);
  low := _TMP_LE3_OUT;
  _TMP_GE31_OUT := GE(EN := TRUE, IN1 := level, IN2 := high_1, ENO => _TMP_GE31_ENO);
  high := _TMP_GE31_OUT;
  pumps := NOT(high) AND (low OR pumps);
  valve := NOT(close_req) AND (valve OR open_req AND NOT(low));
  _TMP_EQ23_OUT := EQ(EN := TRUE, IN1 := request, IN2 := 1, ENO => _TMP_EQ23_ENO);
  open_req := _TMP_EQ23_OUT;
  _TMP_EQ24_OUT := EQ(EN := TRUE, IN1 := request, IN2 := 0, ENO => _TMP_EQ24_ENO);
  close_req := _TMP_EQ24_OUT;
END_PROGRAM

CONFIGURATION Config0

  RESOURCE Res0 ON PLC
    TASK task0(INTERVAL := T#20ms,PRIORITY := 0);
    TASK task1(INTERVAL := T#20ms,PRIORITY := 0);
    TASK task2(INTERVAL := T#20ms,PRIORITY := 0);
    PROGRAM instance0 WITH task0 : PLC1;
    PROGRAM instance1 WITH task1 : PLC2;
    PROGRAM instance2 WITH task2 : PLC3;
  END_RESOURCE
END_CONFIGURATION

(* ---- lb_claude_assisted_973c280d956d_0001.st ---- *)
FUNCTION_BLOCK TONOF

	VAR_INPUT
		IN :	BOOL;
		T_ON :	TIME;
		T_OFF :	TIME;
	END_VAR

	VAR_OUTPUT
		Q :	BOOL;
	END_VAR

	VAR
		X :	TON;
		old :	BOOL;
		mode :	BOOL;
	END_VAR

	IF IN XOR old THEN
	X(IN := FALSE, PT := SEL_TIME(IN,T_OFF,T_ON));
	mode := IN;
	old := IN;
	END_IF;
	X(IN := TRUE);
	IF X.Q THEN Q := mode;END_IF;

END_FUNCTION_BLOCK

FUNCTION UDINT_TO_TIME2:TIME

	VAR_INPUT
		IN :	UDINT;
	END_VAR

	UDINT_TO_TIME2 := DINT_TO_TIME(UDINT_TO_DINT(IN));

END_FUNCTION

FUNCTION_BLOCK T_PLC_MS_block
	VAR_OUTPUT
		T_PLC_MS :	UDINT;
	END_VAR

	VAR_EXTERNAL
		PLC_TICKS_PER_SEC :	INT;
		PLC_SYS_TICK_CNT :	DINT;
	END_VAR

	VAR
		debug :	BOOL;(*Debug-Mode ON / OFF*)
		N :	INT;(*Debug-Faktor*)
		Offset :	UDINT;(*Debug-Offset*)
		temp :	DWORD := DWORD#1;(*Debug-Offset*)
		mode :	BOOL;(*modus*)
		faktor :	UDINT;(*Systemtakt-Faktor*)
		init :	BOOL;
		v_plc_ticks_per_sec :	UDINT;
		base :	UDINT := UDINT#1000;
	END_VAR

	IF init = FALSE THEN
		v_plc_ticks_per_sec := INT_TO_UDINT(PLC_TICKS_PER_SEC);
		IF v_plc_ticks_per_sec = UDINT#1024 THEN
			faktor := UDINT#1;
			mode := FALSE;
		ELSIF v_plc_ticks_per_sec > UDINT#0 THEN
			IF v_plc_ticks_per_sec <= base THEN
				faktor := base / v_plc_ticks_per_sec;
				mode := FALSE;
			ELSE
				faktor := v_plc_ticks_per_sec / base;
				mode := TRUE;
			END_IF;
		ELSE
			faktor := UDINT#1;
		END_IF;
		init := TRUE;
	END_IF;

	IF mode THEN
		T_PLC_MS := DINT_TO_UDINT(PLC_SYS_TICK_CNT) / faktor;
	ELSE
		T_PLC_MS := DINT_TO_UDINT(PLC_SYS_TICK_CNT) * faktor;
	END_IF;

	IF debug THEN
		T_PLC_MS := (DWORD_TO_UDINT(SHL(UDINT_TO_DWORD(T_PLC_MS),N) OR SHL(temp,N)) - UDINT#1) + Offset;
	END_IF;
END_FUNCTION_BLOCK

FUNCTION TIME_TO_UDINT2:UDINT
	VAR_INPUT
		X :	TIME;
	END_VAR

	TIME_TO_UDINT2 := DINT_TO_UDINT(TIME_TO_DINT(X));
END_FUNCTION

FUNCTION_BLOCK ACTUATOR_COIL_Block

	VAR_INPUT
		IN :	BOOL;
		SELF_ACT_CYCLE :	TIME := T#10d;
		SELF_ACT_TIME :	TIME := T#1s;
	END_VAR

	VAR_OUTPUT
		OUT :	BOOL;
		STATUS :	BYTE;
	END_VAR

	VAR
		last :	UDINT;
		init :	BOOL;
		tx :	UDINT;
		now :	UDINT;
		T_PLC_MS :	T_PLC_MS_Block;
	END_VAR

	T_PLC_MS();
	now := T_PLC_MS.T_PLC_MS;

	IF NOT init THEN
		last := now;
		init := TRUE;
	ELSIF IN THEN
		OUT := TRUE;
		STATUS := BYTE#101;
		LAST := now;
	ELSE
		OUT := FALSE;
		STATUS := BYTE#100;
		tx := now - last;
		IF (self_act_cycle > T#0s) AND (tx >= TIME_TO_UDINT2(self_act_cycle)) THEN
			OUT := TRUE;
			STATUS := BYTE#102;
			IF tx >= TIME_TO_UDINT2(self_act_cycle + self_act_time) THEN
				last := now;
				OUT := FALSE;
				STATUS := BYTE#100;
			END_IF;
		END_IF;
	END_IF;

END_FUNCTION_BLOCK

FUNCTION_BLOCK TANK_LEVEL_Block

	VAR_INPUT
		LEVEL :	BOOL;
		LEAK :	BOOL;
		ACLR :	BOOL;
		MAX_VALVE_TIME :	TIME;
		LEVEL_DELAY_TIME :	TIME;
	END_VAR

	VAR_OUTPUT
		VALVE :	BOOL;
		ALARM :	BOOL;
		STATUS :	BYTE;
	END_VAR

	VAR
		cx :	ACTUATOR_COIL_Block;
		tn :	TON;
		tl :	TONOF;
		open :	BOOL;
	END_VAR

	tl(in := level, T_ON := level_delay_time, T_OFF := level_delay_time);
	open := tl.Q;

	IF ALARM THEN
		IF ACLR THEN
			ALARM := FALSE;
			STATUS := BYTE#101;
			cx(in := FALSE);
		END_IF;
		RETURN;
	ELSIF LEAK THEN
		cx(in := FALSE);
		ALARM := TRUE;
		STATUS := BYTE#1;
	ELSIF open THEN
		cx(in := TRUE);
		STATUS := BYTE#102;
	ELSE
		cx(in := FALSE);
		STATUS := BYTE#100;
	END_IF;

	IF open THEN
	    tn(in := cx.out AND (MAX_VALVE_TIME > T#0s), PT := T#9999h);
	ELSE
	    tn(in := cx.out AND (MAX_VALVE_TIME > T#0s), PT := MAX_VALVE_TIME);
	END_IF;
	IF tn.Q THEN
		ALARM := TRUE;
		STATUS := BYTE#2;
		cx(in := FALSE);
	END_IF;

	VALVE := cx.out;
END_FUNCTION_BLOCK

PROGRAM program0
	VAR
		LEVEL :	BOOL;
		LEAK :	BOOL;
		ACLR :	BOOL;
		MAX_VALVE_TIME :	TIME;
		LEVEL_DELAY_TIME :	TIME;
		VALVE :	BOOL;
		ALARM :	BOOL;
		STATUS :	BYTE;

		func_block : TANK_LEVEL_Block;
	END_VAR
	func_block.LEVEL := LEVEL;
	func_block.LEAK := LEAK;
	func_block.ACLR := ACLR ;
	func_block.MAX_VALVE_TIME := MAX_VALVE_TIME;
	func_block.LEVEL_DELAY_TIME := LEVEL_DELAY_TIME ;
	func_block();
	VALVE  := func_block.VALVE;
	ALARM  := func_block.ALARM;
	STATUS  := func_block.STATUS;
END_PROGRAM

CONFIGURATION Config0
	VAR_GLOBAL
		PLC_TICKS_PER_SEC :	INT;
		PLC_SYS_TICK_CNT :	DINT;
	END_VAR
  	RESOURCE Res0 ON PLC
    	TASK task0(INTERVAL := T#20ms,PRIORITY := 0);
    	PROGRAM instance0 WITH task0 : program0;
  	END_RESOURCE
END_CONFIGURATION

(* ---- lb_claude_assisted_9930e0c81d42_0008.st ---- *)
FUNCTION_BLOCK INTERLOCK_Block

	VAR_INPUT
		I1 :	BOOL;
		I2 :	BOOL;
		TL :	TIME;
	END_VAR

	VAR_OUTPUT
		Q1 :	BOOL;
		Q2 :	BOOL;
	END_VAR

	VAR
		T1 :	TOF;
		T2 :	TOF;
	END_VAR

	T1(IN := I1, PT := TL);
	T2(IN := I2, PT := TL);

	Q1 := I1 AND NOT t2.Q;
	Q2 := I2 AND NOT t1.Q;

END_FUNCTION_BLOCK

FUNCTION TIME_TO_UDINT2:UDINT
	VAR_INPUT
		X :	TIME;
	END_VAR

	TIME_TO_UDINT2 := DINT_TO_UDINT(TIME_TO_DINT(X));
END_FUNCTION

FUNCTION_BLOCK T_PLC_MS_block
	VAR_OUTPUT
		T_PLC_MS :	UDINT;
	END_VAR

	VAR_EXTERNAL
		PLC_TICKS_PER_SEC :	INT;
		PLC_SYS_TICK_CNT :	DINT;
	END_VAR

	VAR
		debug :	BOOL;(*Debug-Mode ON / OFF*)
		N :	INT;(*Debug-Faktor*)
		Offset :	UDINT;(*Debug-Offset*)
		temp :	DWORD := DWORD#1;(*Debug-Offset*)
		mode :	BOOL;(*modus*)
		faktor :	UDINT;(*Systemtakt-Faktor*)
		init :	BOOL;
		v_plc_ticks_per_sec :	UDINT;
		base :	UDINT := UDINT#1000;
	END_VAR

	IF init = FALSE THEN
		v_plc_ticks_per_sec := INT_TO_UDINT(PLC_TICKS_PER_SEC);
		IF v_plc_ticks_per_sec = UDINT#1024 THEN
			faktor := UDINT#1;
			mode := FALSE;
		ELSIF v_plc_ticks_per_sec > UDINT#0 THEN
			IF v_plc_ticks_per_sec <= base THEN
				faktor := base / v_plc_ticks_per_sec;
				mode := FALSE;
			ELSE
				faktor := v_plc_ticks_per_sec / base;
				mode := TRUE;
			END_IF;
		ELSE
			faktor := UDINT#1;
		END_IF;
		init := TRUE;
	END_IF;

	IF mode THEN
		T_PLC_MS := DINT_TO_UDINT(PLC_SYS_TICK_CNT) / faktor;
	ELSE
		T_PLC_MS := DINT_TO_UDINT(PLC_SYS_TICK_CNT) * faktor;
	END_IF;

	IF debug THEN
		T_PLC_MS := (DWORD_TO_UDINT(SHL(UDINT_TO_DWORD(T_PLC_MS),N) OR SHL(temp,N)) - UDINT#1) + Offset;
	END_IF;
END_FUNCTION_BLOCK

FUNCTION FRMP_B:BYTE
	VAR_INPUT
		START :	BYTE;
		DIR :	BOOL;
		TD :	TIME;
		TR :	TIME;
	END_VAR

	IF TD < TR THEN
		FRMP_B := MIN(UDINT_TO_BYTE(DWORD_TO_UDINT(SHL(TIME_TO_DWORD(TD), 8)) / TIME_TO_UDINT2(TR)), SEL(DIR, START, USINT_TO_BYTE(USINT#255 - BYTE_TO_USINT(START))));
		IF DIR THEN
			FRMP_B := USINT_TO_BYTE(BYTE_TO_USINT(START) + BYTE_TO_USINT(FRMP_B));
		ELSE
			FRMP_B := USINT_TO_BYTE(BYTE_TO_USINT(START) - BYTE_TO_USINT(FRMP_B));
		END_IF;
	ELSE
		FRMP_B := SEL(DIR, BYTE#0, BYTE#255);
	END_IF;
END_FUNCTION

FUNCTION_BLOCK _RMP_B
	VAR_INPUT
		DIR :	BOOL;
		E :	BOOL := TRUE;
		TR :	TIME;
	END_VAR

	VAR_IN_OUT
		RMP :	BYTE;
	END_VAR

	VAR
		T_PLC_MS :	T_PLC_MS_block;
		tx :	TIME;
		tl :	TIME;
		tn :	TIME;
		init :	BOOL;
		last_dir :	BOOL;
		start :	BYTE;
	END_VAR

	T_PLC_MS();
	tx := UDINT_TO_TIME(T_PLC_MS.T_PLC_MS);

	IF E AND init AND (dir = last_dir) AND (RMP <> SEL(DIR, BYTE#0, BYTE#255)) AND TR = tn THEN
		RMP := FRMP_B(start, DIR, tx - tl, TR);
	ELSE
		init := TRUE;
		tl := tx;
		tn := tr;
		start := RMP;
	END_IF;
	last_dir := dir;
END_FUNCTION_BLOCK

FUNCTION_BLOCK RMP_B_Block

	VAR_INPUT
		SET :	BOOL;
		PT :	TIME;
		E :	BOOL := TRUE;
		UP :	BOOL := TRUE;
		RST :	BOOL;
	END_VAR

	VAR_OUTPUT
		OUT :	BYTE;
		BUSY :	BOOL;
		HIGH :	BOOL;
		LOW :	BOOL;
	END_VAR

	VAR
		rmp :	_RMP_B;
	END_VAR

	rmp(dir := UP, E := E, TR := PT, RMP := out);
	out := rmp.RMP;

	IF RST THEN
		out := BYTE#0;
	ELSIF SET THEN
		out := BYTE#255;
	END_IF;

low := out = BYTE#0;
high := out = BYTE#255;
busy := NOT (low OR high) AND E;

END_FUNCTION_BLOCK

FUNCTION_BLOCK BLIND_ACTUATOR_Block

	VAR_INPUT
		UP :	BOOL;
		DN :	BOOL;
		S_IN :	BYTE;
		T_UD :	TIME := T#10s;
		T_ANGLE :	TIME := T#3s;
		T_LOCKOUT :	TIME := t#100ms;
	END_VAR

	VAR_OUTPUT
		POS :	BYTE;
		ANG :	BYTE;
		QU :	BOOL;
		QD :	BOOL;
		STATUS :	BYTE;
	END_VAR

	VAR
		position :	RMP_B_Block;
		angle :	RMP_B_Block;
		lock :	INTERLOCK_Block;
	END_VAR

	lock(i1 := UP, I2 := DN, TL := T_lockout);

	angle(e := lock.Q1 OR lock.Q2, UP := lock.Q1, PT := T_Angle);
	position(e := lock.Q1 AND angle.high OR lock.Q2 AND angle.low, up := lock.Q1, PT := T_UD);

	pos := position.Out;
	ang := angle.Out;

	QU := lock.Q1;
	QD := lock.Q2;

	IF UP AND DN THEN
		IF UP AND DN THEN
		    status := BYTE#121;
		ELSE
		    status := BYTE#1;
		END_IF;
	ELSIF UP THEN
		status := BYTE#121;
	ELSIF DN THEN
		status := BYTE#122;
	ELSE
		status := S_IN;
	END_IF;

END_FUNCTION_BLOCK

PROGRAM program0
	VAR
		UP :	BOOL;
		DN :	BOOL;
		S_IN :	BYTE;
		T_UD :	TIME := T#10s;
		T_ANGLE :	TIME := T#3s;
		T_LOCKOUT :	TIME := t#100ms;
		POS :	BYTE;
		ANG :	BYTE;
		QU :	BOOL;
		QD :	BOOL;
		func_block : BLIND_ACTUATOR_Block;
	END_VAR
	func_block.UP := UP;
	func_block.DN := DN;
	func_block.S_IN := S_IN ;
	func_block.T_UD := T_UD;
	func_block.T_ANGLE := T_ANGLE;
	func_block.T_LOCKOUT := T_LOCKOUT;
	func_block();
	POS  := func_block.POS;
	ANG  := func_block.ANG;
	QU  := func_block.QU;
	QD  := func_block.QD;
END_PROGRAM

CONFIGURATION Config0
	VAR_GLOBAL
		PLC_TICKS_PER_SEC :	INT;
		PLC_SYS_TICK_CNT :	DINT;
	END_VAR
  	RESOURCE Res0 ON PLC
    	TASK task0(INTERVAL := T#20ms,PRIORITY := 0);
    	PROGRAM instance0 WITH task0 : program0;
  	END_RESOURCE
END_CONFIGURATION

(* ---- lb_claude_assisted_a0c988439d9c_0039.st ---- *)
(*
This code implements a randomly grown symbolic expression:

IN18 | (((xor(xor(xor(xor(IN17 | (xor(xor(IN20 | IN31, !((IN23 | IN3) | (!(IN14)))), xor(xor((!(IN35)) | (!(IN43)), IN8), !(IN28 | IN33)))), false), IN38 & IN24), ((IN39 | (((IN32 | true) | (!(IN47))) | ((xor(xor(IN25, IN42), IN28)) | (IN42 | IN24)))) & ((((xor(xor(IN38, IN18), IN2)) | (IN4 & IN11)) | ((!(IN45)) & (IN8 | IN28))) | (!((!(IN50)) & IN24)))) & (xor(xor(IN18, ((xor(xor(IN35 & IN33, false & IN2), !(IN32))) & (!(IN19 & IN38))) & ((!(xor(xor(IN7, IN2), IN18))) & ((xor(xor(IN48, IN26), false)) & (xor(xor(IN46, IN38), IN13))))), xor(xor(xor(xor(IN13 | (xor(xor(IN37, IN12), IN43)), IN36), xor(xor(IN17 | true, IN49), IN2)), (!(IN33 & IN19)) & IN43), IN7)))), xor(xor(xor(xor(xor(xor(((xor(xor(IN14, IN2), IN34)) & (xor(xor(IN43, IN41), IN11))) | ((IN34 & IN13) | (IN14 & IN33)), !(xor(xor(!(IN26), !(IN28)), !(IN43)))), (xor(xor(IN30, xor(xor(IN38, IN10), IN28)), xor(xor(IN36, IN49), IN11))) | IN9), xor(xor(xor(xor(!(xor(xor(IN48, IN48), IN47)), (!(IN23)) | (IN30 | IN42)), xor(xor(IN21 & IN37, IN19), IN31)), (!(IN28)) | IN38), xor(xor(IN31, !(!(IN19))), IN45))), (xor(xor(IN19, IN15), xor(xor(xor(xor(IN5, IN27), IN1), false), !(IN13)))) & (IN14 & (xor(xor(IN13 & IN11, IN1), xor(xor(true, IN33), IN46))))), IN37), IN6))) | (!(xor(xor((!(((IN13 | IN14) & IN11) | (xor(xor(IN46 & IN42, xor(xor(IN32, IN1), IN3)), !(IN7))))) & IN26, IN17 | IN13), (!(((!(IN34)) & (true & IN40)) & ((xor(xor(IN3, IN6), IN24)) & IN30))) & (((IN21 & (IN16 & IN37)) | (xor(xor(xor(xor(IN47, IN22), IN46), !(IN28)), IN6 | IN26))) | (((xor(xor(IN10, IN47), IN41)) & IN19) | ((!(IN12)) | (!(IN20))))))))) & IN32)

*)

FUNCTION_BLOCK F_CollectInput
  VAR_IN_OUT
      Data : ARRAY[1..50] OF BOOL;
  END_VAR
  VAR_INPUT
      TICK  : BOOL := 0;
      IN1   : BOOL := 0;
      IN2   : BOOL := 0;
      IN3   : BOOL := 0;
      IN4   : BOOL := 0;
      IN5   : BOOL := 0;
      RESET : BOOL := FALSE;
  END_VAR
  VAR_OUTPUT
      Finished : BOOL;
  END_VAR
  VAR
      j    : USINT := 1;
      tock : BOOL  := 0;
  END_VAR
  IF NOT RESET AND tock = NOT TICK THEN
      Data[j]   := IN1;
      Data[j+1] := IN2;
      Data[j+2] := IN3;
      Data[j+3] := IN4;
      Data[j+4] := IN5;
      j := j + 5;
      tock := TICK;
  ELSE
      j := 1;
      tock := 0;
  END_IF;
  Finished := (j > 50);
END_FUNCTION_BLOCK

PROGRAM Boiler
  VAR
    Data  : ARRAY[1..50] OF BOOL;
    Ready : BOOL;
    CollectInput : F_CollectInput;
  END_VAR
  VAR
    TICK     AT %IX1.0 : BOOL;
    IN1      AT %IX0.3 : BOOL;
    IN2      AT %IX0.4 : BOOL;
    IN3      AT %IX0.5 : BOOL;
    IN4      AT %IX0.6 : BOOL;
    IN5      AT %IX0.7 : BOOL;
    OutReady AT %QX0.0 : BOOL := FALSE;
    FeedNext AT %QX0.1 : BOOL := FALSE;
    Out      AT %QX0.2 : BOOL;
  END_VAR
  CollectInput(TICK:=TICK, IN1:=IN1, IN2:=IN2, IN3:=IN3, IN4:=IN4, IN5:=IN5);
  Ready := CollectInput.Finished;
  FeedNext := 1;
  IF Ready THEN
    Out := (Data[18] OR (((((((Data[17] OR (((Data[20] OR Data[31]) XOR (NOT ((Data[23] OR Data[3]) OR (NOT Data[14])))) XOR ((((NOT Data[35]) OR (NOT Data[43])) XOR Data[8]) XOR (NOT (Data[28] OR Data[33]))))) XOR FALSE) XOR (Data[38] AND Data[24])) XOR (((Data[39] OR (((Data[32] OR TRUE) OR (NOT Data[47])) OR (((Data[25] XOR Data[42]) XOR Data[28]) OR (Data[42] OR Data[24])))) AND (((((Data[38] XOR Data[18]) XOR Data[2]) OR (Data[4] AND Data[11])) OR ((NOT Data[45]) AND (Data[8] OR Data[28]))) OR (NOT ((NOT Data[50]) AND Data[24])))) AND ((Data[18] XOR (((((Data[35] AND Data[33]) XOR (FALSE AND Data[2])) XOR (NOT Data[32])) AND (NOT (Data[19] AND Data[38]))) AND ((NOT ((Data[7] XOR Data[2]) XOR Data[18])) AND (((Data[48] XOR Data[26]) XOR FALSE) AND ((Data[46] XOR Data[38]) XOR Data[13]))))) XOR (((((Data[13] OR ((Data[37] XOR Data[12]) XOR Data[43])) XOR Data[36]) XOR (((Data[17] OR TRUE) XOR Data[49]) XOR Data[2])) XOR ((NOT (Data[33] AND Data[19])) AND Data[43])) XOR Data[7])))) XOR ((((((((((Data[14] XOR Data[2]) XOR Data[34]) AND ((Data[43] XOR Data[41]) XOR Data[11])) OR ((Data[34] AND Data[13]) OR (Data[14] AND Data[33]))) XOR (NOT (((NOT Data[26]) XOR (NOT Data[28])) XOR (NOT Data[43])))) XOR (((Data[30] XOR ((Data[38] XOR Data[10]) XOR Data[28])) XOR ((Data[36] XOR Data[49]) XOR Data[11])) OR Data[9])) XOR (((((NOT ((Data[48] XOR Data[48]) XOR Data[47])) XOR ((NOT Data[23]) OR (Data[30] OR Data[42]))) XOR (((Data[21] AND Data[37]) XOR Data[19]) XOR Data[31])) XOR ((NOT Data[28]) OR Data[38])) XOR ((Data[31] XOR (NOT (NOT Data[19]))) XOR Data[45]))) XOR (((Data[19] XOR Data[15]) XOR ((((Data[5] XOR Data[27]) XOR Data[1]) XOR FALSE) XOR (NOT Data[13]))) AND (Data[14] AND (((Data[13] AND Data[11]) XOR Data[1]) XOR ((TRUE XOR Data[33]) XOR Data[46]))))) XOR Data[37]) XOR Data[6])) OR (NOT ((((NOT (((Data[13] OR Data[14]) AND Data[11]) OR (((Data[46] AND Data[42]) XOR ((Data[32] XOR Data[1]) XOR Data[3])) XOR (NOT Data[7])))) AND Data[26]) XOR (Data[17] OR Data[13])) XOR ((NOT (((NOT Data[34]) AND (TRUE AND Data[40])) AND (((Data[3] XOR Data[6]) XOR Data[24]) AND Data[30]))) AND (((Data[21] AND (Data[16] AND Data[37])) OR ((((Data[47] XOR Data[22]) XOR Data[46]) XOR (NOT Data[28])) XOR (Data[6] OR Data[26]))) OR ((((Data[10] XOR Data[47]) XOR Data[41]) AND Data[19]) OR ((NOT Data[12]) OR (NOT Data[20])))))))) AND Data[32]));
    IF Ready THEN
        OutReady := 0;
    ELSE
        OutReady := 1;
    END_IF;
    CollectInput(RESET:=TRUE);
  END_IF;
END_PROGRAM

CONFIGURATION Config0
  RESOURCE Res0 ON PLC
    TASK task0(INTERVAL := T#20ms,PRIORITY := 0);
    PROGRAM instance0 WITH task0 : Boiler;
  END_RESOURCE
END_CONFIGURATION

(* ---- lb_claude_assisted_a0f84c9668d2_0129.st ---- *)
FUNCTION_BLOCK T_PLC_MS_block
	VAR_OUTPUT
		T_PLC_MS :	UDINT;
	END_VAR

	VAR_EXTERNAL
		PLC_TICKS_PER_SEC :	INT;
		PLC_SYS_TICK_CNT :	DINT;
	END_VAR

	VAR
		debug :	BOOL;(*Debug-Mode ON / OFF*)
		N :	INT;(*Debug-Faktor*)
		Offset :	UDINT;(*Debug-Offset*)
		temp :	DWORD := DWORD#1;(*Debug-Offset*)
		mode :	BOOL;(*modus*)
		faktor :	UDINT;(*Systemtakt-Faktor*)
		init :	BOOL;
		v_plc_ticks_per_sec :	UDINT;
		base :	UDINT := UDINT#1000;
	END_VAR

	IF init = FALSE THEN
		v_plc_ticks_per_sec := INT_TO_UDINT(PLC_TICKS_PER_SEC);
		IF v_plc_ticks_per_sec = UDINT#1024 THEN
			faktor := UDINT#1;
			mode := FALSE;
		ELSIF v_plc_ticks_per_sec > UDINT#0 THEN
			IF v_plc_ticks_per_sec <= base THEN
				faktor := base / v_plc_ticks_per_sec;
				mode := FALSE;
			ELSE
				faktor := v_plc_ticks_per_sec / base;
				mode := TRUE;
			END_IF;
		ELSE
			faktor := UDINT#1;
		END_IF;
		init := TRUE;
	END_IF;

	IF mode THEN
		IF mode THEN
		    T_PLC_MS := DINT_TO_UDINT(PLC_SYS_TICK_CNT) * faktor;
		ELSE
		    T_PLC_MS := DINT_TO_UDINT(PLC_SYS_TICK_CNT) / faktor;
		END_IF;
	ELSE
		T_PLC_MS := DINT_TO_UDINT(PLC_SYS_TICK_CNT) * faktor;
	END_IF;

	IF debug THEN
		T_PLC_MS := (DWORD_TO_UDINT(SHL(UDINT_TO_DWORD(T_PLC_MS),N) OR SHL(temp,N)) - UDINT#1) + Offset;
	END_IF;
END_FUNCTION_BLOCK

FUNCTION_BLOCK FT_RMP

	VAR_INPUT
		RMP :	BOOL := TRUE;
		IN :	REAL;
		KR :	REAL;
		KF :	REAL;
	END_VAR

	VAR_OUTPUT
		OUT :	REAL;
		BUSY :	BOOL;
		UD :	BOOL;
	END_VAR

	VAR
		tx :	TIME;
		last :	TIME;
		init :	BOOL;
		T_PLC_MS :	T_PLC_MS_block;
	END_VAR

	T_PLC_MS();
	tx:= UDINT_TO_TIME(T_PLC_MS.T_PLC_MS) - last;

	IF NOT init THEN
		init := TRUE;
		last := tx;
		tx := t#0s;
		out := in;
	END_IF;
	IF NOT rmp THEN
		out := in;
		busy := FALSE;
	ELSIF out > in THEN
		(* ramp down *)
		out := out - TIME_TO_REAL(tx) * 0.001 * KF;
		out := MAX(in, out);
	ELSIF out < in THEN
		(* ramp up *)
		out := out + TIME_TO_REAL(tx) * 0.001 * KR;
		out := MIN(in, out);
	END_IF;

	(* set busy and dir flags *)
	IF out < in THEN
		busy := TRUE;
		ud := TRUE;
	ELSIF out > in THEN
		busy := TRUE;
		ud := FALSE;
	ELSE
		busy := FALSE;
	END_IF;
	last := last + tx;

END_FUNCTION_BLOCK

PROGRAM program0
	VAR
		RMP :	BOOL := TRUE;
		IN :	REAL;
		KR :	REAL;
		KF :	REAL;

		OUT :	REAL;
		BUSY :	BOOL;
		UD :	BOOL;

		func_block : FT_RMP;
	END_VAR
	func_block.RMP := RMP;
	func_block.IN := IN;
	func_block.KR := KR;
	func_block.KF := KF;
	func_block();
	OUT := func_block.OUT;
	BUSY := func_block.BUSY;
	UD := func_block.UD;

END_PROGRAM

CONFIGURATION Config0

	VAR_GLOBAL
		PLC_TICKS_PER_SEC :	INT;
		PLC_SYS_TICK_CNT :	DINT;
	END_VAR

	RESOURCE Res0 ON PLC
		TASK task0(INTERVAL := T#20ms,PRIORITY := 0);
		PROGRAM instance0 WITH task0 : program0;
	END_RESOURCE

END_CONFIGURATION

(* ---- lb_claude_assisted_a2db08096301_0037.st ---- *)
(*
This code implements a randomly grown symbolic expression:

((xor(xor(xor(xor(xor(xor(IN48, xor(xor((!((xor(xor(IN5, IN42), IN45)) | (IN37 & false))) & (xor(xor(xor(xor(IN2, !(IN14)), IN48), xor(xor(IN21 | IN17, IN27 | IN19), IN36)), !(IN13 & IN45))), IN27), ((!(xor(xor(IN17, IN29), IN43))) & ((xor(xor(IN39, IN3), IN34)) | IN14)) & ((!(xor(xor(IN39, IN41), IN17))) & true))), IN46), !(!((IN43 & ((xor(xor(IN37, IN8), IN48)) & (IN16 & IN16))) & (!((IN15 | IN18) | IN37))))), (xor(xor(!(IN34 & (xor(xor(IN9 & IN18, xor(xor(false, IN44), IN30)), IN5))), xor(xor(((!(IN48)) | (IN17 & IN37)) | IN1, !((xor(xor(IN10, IN18), IN41)) | (IN45 & IN13))), IN4 | (!(IN41 & IN27)))), !((!(IN7 | IN36)) & ((!(IN20)) | IN9)))) | ((!(!(IN29))) | IN6)), IN2), xor(xor(IN43 | (xor(xor(((xor(xor(!(IN14), !(IN15)), xor(xor(IN1, IN15), IN50))) & ((IN10 & IN6) & (IN6 | IN7))) | (!((IN15 | IN26) | (!(IN41)))), xor(xor(!(!(!(IN43))), IN36 & IN15), IN31 | (IN42 & (IN48 & IN47)))), ((xor(xor(!(IN23), IN15 & IN10), IN31)) & (xor(xor(xor(xor(IN29, IN46), false), IN15), !(IN7)))) & IN24)), xor(xor(IN5, IN16), !((!(!(xor(xor(IN10, IN47), IN10)))) | (IN8 | ((!(IN18)) | (!(IN31))))))), (true | ((!(xor(xor(IN20 | IN43, IN4 & IN11), !(IN3)))) | (IN17 | (!(IN28 | IN3))))) | ((!(!((IN18 | IN37) & (xor(xor(IN12, IN43), IN4))))) & IN23)))) & ((!(IN17)) & (!(IN45)))) | (IN33 & (xor(xor(!(IN17), xor(xor(!((xor(xor(!(!(!(IN39))), xor(xor(!(IN13 & IN33), IN33 | IN16), (xor(xor(IN3, IN11), IN19)) & (IN6 | IN22))), ((IN18 & IN3) | (IN40 | IN23)) | ((IN41 | true) & IN44))) & IN13), (!(IN9 & (((!(IN38)) | (true & IN36)) & IN38))) & (!(((!(!(IN46))) & ((IN15 & IN28) & (IN16 | IN9))) & ((xor(xor(IN7, !(IN13)), IN41 & IN6)) | (xor(xor(xor(xor(IN40, IN31), IN6), !(IN39)), !(IN46))))))), IN11)), IN35)))

*)

FUNCTION_BLOCK F_CollectInput
  VAR_IN_OUT
      Data : ARRAY[1..50] OF BOOL;
  END_VAR
  VAR_INPUT
      TICK  : BOOL := 0;
      IN1   : BOOL := 0;
      IN2   : BOOL := 0;
      IN3   : BOOL := 0;
      IN4   : BOOL := 0;
      IN5   : BOOL := 0;
      RESET : BOOL := FALSE;
  END_VAR
  VAR_OUTPUT
      Finished : BOOL;
  END_VAR
  VAR
      j    : USINT := 1;
      tock : BOOL  := 0;
  END_VAR
  IF NOT RESET AND tock = NOT TICK THEN
      Data[j]   := IN1;
      Data[j+1] := IN2;
      Data[j+2] := IN3;
      Data[j+3] := IN4;
      Data[j+4] := IN5;
      j := j + 5;
      tock := TICK;
  ELSE
      j := 1;
      tock := 0;
  END_IF;
  Finished := (j > 50);
END_FUNCTION_BLOCK

PROGRAM Boiler
  VAR
    Data  : ARRAY[1..50] OF BOOL;
    Ready : BOOL;
    CollectInput : F_CollectInput;
  END_VAR
  VAR
    TICK     AT %IX1.0 : BOOL;
    IN1      AT %IX0.3 : BOOL;
    IN2      AT %IX0.4 : BOOL;
    IN3      AT %IX0.5 : BOOL;
    IN4      AT %IX0.6 : BOOL;
    IN5      AT %IX0.7 : BOOL;
    OutReady AT %QX0.0 : BOOL := FALSE;
    FeedNext AT %QX0.1 : BOOL := FALSE;
    Out      AT %QX0.2 : BOOL;
  END_VAR
  CollectInput(TICK:=TICK, IN1:=IN1, IN2:=IN2, IN3:=IN3, IN4:=IN4, IN5:=IN5);
  Ready := CollectInput.Finished;
  FeedNext := 1;
  IF Ready THEN
    Out := ((((((((Data[48] XOR ((((NOT (((Data[5] XOR Data[42]) XOR Data[45]) OR (Data[37] AND FALSE))) AND ((((Data[2] XOR (NOT Data[14])) XOR Data[48]) XOR (((Data[21] OR Data[17]) XOR (Data[27] OR Data[19])) XOR Data[36])) XOR (NOT (Data[13] AND Data[45])))) XOR Data[27]) XOR (((NOT ((Data[17] XOR Data[29]) XOR Data[43])) AND (((Data[39] XOR Data[3]) XOR Data[34]) OR Data[14])) AND ((NOT ((Data[39] XOR Data[41]) XOR Data[17])) AND TRUE)))) XOR Data[46]) XOR (NOT (NOT ((Data[43] AND (((Data[37] XOR Data[8]) XOR Data[48]) AND (Data[16] AND Data[16]))) AND (NOT ((Data[15] OR Data[18]) OR Data[37])))))) XOR ((((NOT (Data[34] AND (((Data[9] AND Data[18]) XOR ((FALSE XOR Data[44]) XOR Data[30])) XOR Data[5]))) XOR (((((NOT Data[48]) OR (Data[17] AND Data[37])) OR Data[1]) XOR (NOT (((Data[10] XOR Data[18]) XOR Data[41]) OR (Data[45] AND Data[13])))) XOR (Data[4] OR (NOT (Data[41] AND Data[27]))))) XOR (NOT ((NOT (Data[7] OR Data[36])) AND ((NOT Data[20]) OR Data[9])))) OR ((NOT (NOT Data[29])) OR Data[6]))) XOR Data[2]) XOR (((Data[43] OR (((((((NOT Data[14]) XOR (NOT Data[15])) XOR ((Data[1] XOR Data[15]) XOR Data[50])) AND ((Data[10] AND Data[6]) AND (Data[6] OR Data[7]))) OR (NOT ((Data[15] OR Data[26]) OR (NOT Data[41])))) XOR (((NOT (NOT (NOT Data[43]))) XOR (Data[36] AND Data[15])) XOR (Data[31] OR (Data[42] AND (Data[48] AND Data[47]))))) XOR (((((NOT Data[23]) XOR (Data[15] AND Data[10])) XOR Data[31]) AND ((((Data[29] XOR Data[46]) XOR FALSE) XOR Data[15]) XOR (NOT Data[7]))) AND Data[24]))) XOR ((Data[5] XOR Data[16]) XOR (NOT ((NOT (NOT ((Data[10] XOR Data[47]) XOR Data[10]))) OR (Data[8] OR ((NOT Data[18]) OR (NOT Data[31]))))))) XOR ((TRUE OR ((NOT (((Data[20] OR Data[43]) XOR (Data[4] AND Data[11])) XOR (NOT Data[3]))) OR (Data[17] OR (NOT (Data[28] OR Data[3]))))) OR ((NOT (NOT ((Data[18] OR Data[37]) AND ((Data[12] XOR Data[43]) XOR Data[4])))) AND Data[23])))) AND ((NOT Data[17]) AND (NOT Data[45]))) OR (Data[33] AND (((NOT Data[17]) XOR (((NOT ((((NOT (NOT (NOT Data[39]))) XOR (((NOT (Data[13] AND Data[33])) XOR (Data[33] OR Data[16])) XOR (((Data[3] XOR Data[11]) XOR Data[19]) AND (Data[6] OR Data[22])))) XOR (((Data[18] AND Data[3]) OR (Data[40] OR Data[23])) OR ((Data[41] OR TRUE) AND Data[44]))) AND Data[13])) XOR ((NOT (Data[9] AND (((NOT Data[38]) OR (TRUE AND Data[36])) AND Data[38]))) AND (NOT (((NOT (NOT Data[46])) AND ((Data[15] AND Data[28]) AND (Data[16] OR Data[9]))) AND (((Data[7] XOR (NOT Data[13])) XOR (Data[41] AND Data[6])) OR ((((Data[40] XOR Data[31]) XOR Data[6]) XOR (NOT Data[39])) XOR (NOT Data[46]))))))) XOR Data[11])) XOR Data[35])));
    IF Ready THEN
        OutReady := 0;
    ELSE
        OutReady := 1;
    END_IF;
    CollectInput(RESET:=TRUE);
  END_IF;
END_PROGRAM

CONFIGURATION Config0
  RESOURCE Res0 ON PLC
    TASK task0(INTERVAL := T#20ms,PRIORITY := 0);
    PROGRAM instance0 WITH task0 : Boiler;
  END_RESOURCE
END_CONFIGURATION

(* ---- lb_claude_assisted_a32dad9bc33a_0015.st ---- *)
(*
This code implements a randomly grown symbolic expression:

xor(xor(!(xor(xor(IN32, (!(!((IN49 | (!(IN19))) & (!(IN28 & (xor(xor(IN18, IN20), IN24))))))) & ((xor(xor(IN13, IN1), !(xor(xor(xor(xor(!(IN32), IN20 & IN18), IN50 & IN1), (IN10 & IN17) & (IN11 & IN39)), true & IN1)))) | (xor(xor((!(IN35)) | IN42, !(IN44 | ((!(IN28)) | IN34))), (!((xor(xor(IN28, IN8), IN8)) & IN14)) | (!(xor(xor(xor(xor(IN16, IN9), IN43), xor(xor(IN30, IN9), IN40)), IN50 | IN28))))))), xor(xor((xor(xor(!(((!(IN18)) & (!(IN40))) & (IN28 & (!(IN19)))), IN7), (!((xor(xor(IN34, IN23), IN2)) & (xor(xor(IN27, IN44), IN31)))) | (!(xor(xor(!(IN25), IN8 & IN22), IN9))))) & (xor(xor(IN3, (!(IN42)) & (xor(xor(xor(xor(IN29 & IN50, IN38 | IN40), !(IN36)), IN40), (!(IN24)) & false))), (((!(IN11)) | (!(IN14))) | ((!(IN10)) | (IN36 & IN47))) | IN15)), (!(!(IN45))) & (xor(xor(IN31 | true, IN38), xor(xor(IN43, xor(xor(IN1, (IN12 & IN45) | (IN48 | IN6)), xor(xor(xor(xor(IN28, IN15), IN16), IN6), !(IN49)))), IN13 | ((xor(xor(IN45, IN5), IN32)) & (xor(xor(IN49, IN26), IN28))))))), !((!(IN43)) | (IN45 | (IN20 & (!(xor(xor(IN16, IN7), IN9))))))))), xor(xor((IN15 & ((!(xor(xor(!(xor(xor(IN18 | IN27, xor(xor(IN38, IN31), IN37)), !(IN3))), IN8 & (!(IN28 | IN17))), (xor(xor(IN17 | IN48, xor(xor(IN42, true), true)), IN31 | IN45)) | (IN25 | (!(IN12)))))) | ((!((xor(xor(!(IN16), IN16), xor(xor(IN32, IN22), IN35))) | IN22)) & ((!(xor(xor(IN8, xor(xor(IN18, IN44), IN32)), IN10 | IN3))) & (IN48 & (IN40 | (IN42 & IN27))))))) & IN10, ((!(!(xor(xor(IN3, IN47), (!(IN36 & IN49)) | ((xor(xor(IN42, IN21), IN34)) | (xor(xor(IN24, IN27), IN13))))))) | ((!(IN3)) & IN11)) & (!(((xor(xor(IN31 & IN15, ((!(IN49)) & (xor(xor(IN42, IN39), IN29))) & IN5), (IN7 | (IN32 | IN49)) & ((!(IN32)) | IN44))) & (!(!(!(IN47 & IN34))))) | (((true | (xor(xor(!(IN5), IN9 | IN38), !(IN46)))) | (!((IN37 | IN29) | (IN12 & IN37)))) | IN9)))), !((xor(xor(xor(xor(!(IN20), IN29 | IN30), (xor(xor(IN2, (IN21 & IN3) | (IN13 | IN7)), IN28)) | (xor(xor(IN44, IN21), (!(IN49)) & (!(IN44))))), xor(xor(xor(xor(xor(xor((!(IN48)) & (xor(xor(IN4, IN4), IN39)), (IN31 & IN45) & (IN44 | IN11)), IN5), IN42 & IN13), xor(xor(IN42, (xor(xor(IN14, IN11), IN43)) & IN1), true & (!(IN29)))), !(IN20)), true | (((xor(xor(IN15, IN17), IN17)) | IN20) | (!(!(IN29)))))), (!(IN1 | (xor(xor(IN14 & IN10, !(IN14)), IN21 & IN34)))) & IN17)) | ((IN1 & (xor(xor((!(IN2 & IN15)) | IN22, (!(IN21)) | (IN15 & IN29)), !(xor(xor(IN40, IN7 & IN9), IN31))))) & (((((IN44 & IN35) & (!(IN27))) | IN14) & (IN31 | ((!(IN25)) | (!(IN45))))) | (IN34 | (!((IN22 | IN16) & IN33)))))))), !(IN31 & ((!(xor(xor(((xor(xor(IN2 & IN9, IN28 & IN31), !(IN12))) | ((IN37 | IN35) | IN39)) | ((xor(xor(IN39 & IN49, IN2), IN26 | IN19)) | IN2), xor(xor((IN41 & (!(IN16))) & (xor(xor(!(IN33), IN12 & IN24), IN29 & IN35)), ((IN50 | IN17) & (IN41 & IN40)) | IN5), xor(xor(true, xor(xor(!(IN50), xor(xor(IN37, IN38), IN12)), !(IN47))), !(IN11 | IN42)))), IN42 | IN28))) | ((IN38 & IN43) & IN36))))

*)

FUNCTION_BLOCK F_CollectInput
  VAR_IN_OUT
      Data : ARRAY[1..50] OF BOOL;
  END_VAR
  VAR_INPUT
      TICK  : BOOL := 0;
      IN1   : BOOL := 0;
      IN2   : BOOL := 0;
      IN3   : BOOL := 0;
      IN4   : BOOL := 0;
      IN5   : BOOL := 0;
      RESET : BOOL := FALSE;
  END_VAR
  VAR_OUTPUT
      Finished : BOOL;
  END_VAR
  VAR
      j    : USINT := 1;
      tock : BOOL  := 0;
  END_VAR
  IF NOT RESET AND tock = NOT TICK THEN
      Data[j]   := IN1;
      Data[j+1] := IN2;
      Data[j+2] := IN3;
      Data[j+3] := IN4;
      Data[j+4] := IN5;
      j := j + 5;
      tock := TICK;
  ELSE
      j := 1;
      tock := 0;
  END_IF;
  Finished := (j > 50);
END_FUNCTION_BLOCK

PROGRAM Boiler
  VAR
    Data  : ARRAY[1..50] OF BOOL;
    Ready : BOOL;
    CollectInput : F_CollectInput;
  END_VAR
  VAR
    TICK     AT %IX1.0 : BOOL;
    IN1      AT %IX0.3 : BOOL;
    IN2      AT %IX0.4 : BOOL;
    IN3      AT %IX0.5 : BOOL;
    IN4      AT %IX0.6 : BOOL;
    IN5      AT %IX0.7 : BOOL;
    OutReady AT %QX0.0 : BOOL := FALSE;
    FeedNext AT %QX0.1 : BOOL := FALSE;
    Out      AT %QX0.2 : BOOL;
  END_VAR
  CollectInput(TICK:=TICK, IN1:=IN1, IN2:=IN2, IN3:=IN3, IN4:=IN4, IN5:=IN5);
  Ready := CollectInput.Finished;
  FeedNext := 1;
  IF Ready THEN
    Out := (((NOT ((Data[32] XOR ((NOT (NOT ((Data[49] OR (NOT Data[19])) AND (NOT (Data[28] AND ((Data[18] XOR Data[20]) XOR Data[24])))))) AND (((Data[13] XOR Data[1]) XOR (NOT (((((NOT Data[32]) XOR (Data[20] AND Data[18])) XOR (Data[50] AND Data[1])) XOR ((Data[10] AND Data[17]) AND (Data[11] AND Data[39]))) XOR (TRUE AND Data[1])))) OR ((((NOT Data[35]) OR Data[42]) XOR (NOT (Data[44] OR ((NOT Data[28]) OR Data[34])))) XOR ((NOT (((Data[28] XOR Data[8]) XOR Data[8]) AND Data[14])) OR (NOT ((((Data[16] XOR Data[9]) XOR Data[43]) XOR ((Data[30] XOR Data[9]) XOR Data[40])) XOR (Data[50] OR Data[28])))))))) XOR ((((((NOT (((NOT Data[18]) AND (NOT Data[40])) AND (Data[28] AND (NOT Data[19])))) XOR Data[7]) XOR ((NOT (((Data[34] XOR Data[23]) XOR Data[2]) AND ((Data[27] XOR Data[44]) XOR Data[31]))) OR (NOT (((NOT Data[25]) XOR (Data[8] AND Data[22])) XOR Data[9])))) AND ((Data[3] XOR ((NOT Data[42]) AND (((((Data[29] AND Data[50]) XOR (Data[38] OR Data[40])) XOR (NOT Data[36])) XOR Data[40]) XOR ((NOT Data[24]) AND FALSE)))) XOR ((((NOT Data[11]) OR (NOT Data[14])) OR ((NOT Data[10]) OR (Data[36] AND Data[47]))) OR Data[15]))) XOR ((NOT (NOT Data[45])) AND (((Data[31] OR TRUE) XOR Data[38]) XOR ((Data[43] XOR ((Data[1] XOR ((Data[12] AND Data[45]) OR (Data[48] OR Data[6]))) XOR ((((Data[28] XOR Data[15]) XOR Data[16]) XOR Data[6]) XOR (NOT Data[49])))) XOR (Data[13] OR (((Data[45] XOR Data[5]) XOR Data[32]) AND ((Data[49] XOR Data[26]) XOR Data[28]))))))) XOR (NOT ((NOT Data[43]) OR (Data[45] OR (Data[20] AND (NOT ((Data[16] XOR Data[7]) XOR Data[9]))))))))) XOR ((((Data[15] AND ((NOT (((NOT (((Data[18] OR Data[27]) XOR ((Data[38] XOR Data[31]) XOR Data[37])) XOR (NOT Data[3]))) XOR (Data[8] AND (NOT (Data[28] OR Data[17])))) XOR ((((Data[17] OR Data[48]) XOR ((Data[42] XOR TRUE) XOR TRUE)) XOR (Data[31] OR Data[45])) OR (Data[25] OR (NOT Data[12]))))) OR ((NOT ((((NOT Data[16]) XOR Data[16]) XOR ((Data[32] XOR Data[22]) XOR Data[35])) OR Data[22])) AND ((NOT ((Data[8] XOR ((Data[18] XOR Data[44]) XOR Data[32])) XOR (Data[10] OR Data[3]))) AND (Data[48] AND (Data[40] OR (Data[42] AND Data[27]))))))) AND Data[10]) XOR (((NOT (NOT ((Data[3] XOR Data[47]) XOR ((NOT (Data[36] AND Data[49])) OR (((Data[42] XOR Data[21]) XOR Data[34]) OR ((Data[24] XOR Data[27]) XOR Data[13])))))) OR ((NOT Data[3]) AND Data[11])) AND (NOT (((((Data[31] AND Data[15]) XOR (((NOT Data[49]) AND ((Data[42] XOR Data[39]) XOR Data[29])) AND Data[5])) XOR ((Data[7] OR (Data[32] OR Data[49])) AND ((NOT Data[32]) OR Data[44]))) AND (NOT (NOT (NOT (Data[47] AND Data[34]))))) OR (((TRUE OR (((NOT Data[5]) XOR (Data[9] OR Data[38])) XOR (NOT Data[46]))) OR (NOT ((Data[37] OR Data[29]) OR (Data[12] AND Data[37])))) OR Data[9]))))) XOR (NOT ((((((NOT Data[20]) XOR (Data[29] OR Data[30])) XOR (((Data[2] XOR ((Data[21] AND Data[3]) OR (Data[13] OR Data[7]))) XOR Data[28]) OR ((Data[44] XOR Data[21]) XOR ((NOT Data[49]) AND (NOT Data[44]))))) XOR ((((((((NOT Data[48]) AND ((Data[4] XOR Data[4]) XOR Data[39])) XOR ((Data[31] AND Data[45]) AND (Data[44] OR Data[11]))) XOR Data[5]) XOR (Data[42] AND Data[13])) XOR ((Data[42] XOR (((Data[14] XOR Data[11]) XOR Data[43]) AND Data[1])) XOR (TRUE AND (NOT Data[29])))) XOR (NOT Data[20])) XOR (TRUE OR ((((Data[15] XOR Data[17]) XOR Data[17]) OR Data[20]) OR (NOT (NOT Data[29])))))) XOR ((NOT (Data[1] OR (((Data[14] AND Data[10]) XOR (NOT Data[14])) XOR (Data[21] AND Data[34])))) AND Data[17])) OR ((Data[1] AND ((((NOT (Data[2] AND Data[15])) OR Data[22]) XOR ((NOT Data[21]) OR (Data[15] AND Data[29]))) XOR (NOT ((Data[40] XOR (Data[7] AND Data[9])) XOR Data[31])))) AND (((((Data[44] AND Data[35]) AND (NOT Data[27])) OR Data[14]) AND (Data[31] OR ((NOT Data[25]) OR (NOT Data[45])))) OR (Data[34] OR (NOT ((Data[22] OR Data[16]) AND Data[33]))))))))) XOR (NOT (Data[31] AND ((NOT (((((((Data[2] AND Data[9]) XOR (Data[28] AND Data[31])) XOR (NOT Data[12])) OR ((Data[37] OR Data[35]) OR Data[39])) OR ((((Data[39] AND Data[49]) XOR Data[2]) XOR (Data[26] OR Data[19])) OR Data[2])) XOR ((((Data[41] AND (NOT Data[16])) AND (((NOT Data[33]) XOR (Data[12] AND Data[24])) XOR (Data[29] AND Data[35]))) XOR (((Data[50] OR Data[17]) AND (Data[41] AND Data[40])) OR Data[5])) XOR ((TRUE XOR (((NOT Data[50]) XOR ((Data[37] XOR Data[38]) XOR Data[12])) XOR (NOT Data[47]))) XOR (NOT (Data[11] OR Data[42]))))) XOR (Data[42] OR Data[28]))) OR ((Data[38] AND Data[43]) AND Data[36])))));
    IF Ready THEN
        OutReady := 0;
    ELSE
        OutReady := 1;
    END_IF;
    CollectInput(RESET:=TRUE);
  END_IF;
END_PROGRAM

CONFIGURATION Config0
  RESOURCE Res0 ON PLC
    TASK task0(INTERVAL := T#20ms,PRIORITY := 0);
    PROGRAM instance0 WITH task0 : Boiler;
  END_RESOURCE
END_CONFIGURATION

(* ---- lb_claude_assisted_a7b47d14d4a9_0006.st ---- *)
FUNCTION_BLOCK FLOW_CONTROL_4
	VAR_INPUT
		I0 :	BOOL;
		I1 :	BOOL;
		I2 :	BOOL;
		I3 :	BOOL;
		PR :	BOOL;
		ICE :	BOOL;
		DIAG :	BOOL;
		ENQ :	BOOL;
		RST :	BOOL := FALSE;
		TD_WAIT :	TIME := T#5s;
		TD_S :	TIME := T#10s;
		TD_0 :	TIME := T#10s;
	END_VAR

	VAR_OUTPUT
		QS :	BOOL;
		Q0 :	BOOL;
		Q1 :	BOOL;
		Q2 :	BOOL;
		Q3 :	BOOL;
		ERROR :	BOOL;
		STATUS :	BYTE;
	END_VAR

	VAR
		state :	INT;
		timer :	TP;
	END_VAR

	IF RST THEN
		STATUS := BYTE#100;
		state := 0;
		ERROR := FALSE;

	ELSIF DIAG THEN
		CASE state OF
			0 : (* START diag operation *)
				(* close all VALVEs and pressurize the system *)
				QS := TRUE;
				Q0 := FALSE;
				Q1 := FALSE;
				Q2 := FALSE;
				Q3 := FALSE;
				IF DIAG THEN
				    timer(IN := TRUE, PT := T#9999h);
				ELSE
				    timer(IN := TRUE, PT := TD_WAIT);
				END_IF;
				timer.IN := FALSE;
				state := 1;
			1 : (* wait for TD_wait *)
				timer();
				IF NOT timer.Q THEN
					QS := FALSE;
					timer(IN := TRUE, PT := TD_S);
					timer.IN := FALSE;
					state := 2;
				END_IF;
			2:	(* wait for safety VALVE pressure test *)
				timer();
				IF NOT timer.Q THEN
					IF NOT PR THEN
						(* system pressure failure *)
						ERROR := TRUE;
						STATUS := BYTE#1;
						RETURN;
					END_IF;
					timer(IN := TRUE, PT := TD_0);
					timer.IN := FALSE;
					Q0 := TRUE;
					state := 3;
				END_IF;
			3:	(* wait for pressure on Q0 to hold TD_0 *)
				timer();
				IF NOT timer.Q THEN
					IF NOT PR THEN
						(* VALVE 0 pressure failure *)
						ERROR := TRUE;
						STATUS := BYTE#1;
						RETURN;
					END_IF;
					Q0 := FALSE;
					QS := TRUE;
				END_IF;
		END_CASE;
	ELSIF ICE THEN
		(* when frost is present we close the safety VALVE and open all other VALVEs to depressurize the VALVEs *)
		QS := FALSE;
		Q0 := TRUE;
		Q1 := TRUE;
		Q2 := TRUE;
		Q3 := TRUE;
		STATUS := BYTE#110;

	ELSIF NOT ERROR AND ENQ THEN
			Q0 := I0;
			Q1 := I1;
			Q2 := I2;
			Q3 := I3;
			QS := Q0 OR Q1 OR Q2 OR Q3;
			STATUS := BYTE#100;

			(* maximum ontime check *)
	ELSE
		Q0 := FALSE;
		Q1 := FALSE;
		Q2 := FALSE;
		Q3 := FALSE;
	END_IF;

END_FUNCTION_BLOCK

PROGRAM program0
  VAR
		I0   :	BOOL;
		I1   :	BOOL;
		I2   :	BOOL;
		I3   :	BOOL;
		PR   :	BOOL;
		ICE  :	BOOL;
		DIAG :	BOOL;
		ENQ  :	BOOL;
		RST  :	BOOL ;
		TD_WAIT :	TIME;
		TD_S    :	TIME;
		TD_0    :	TIME;

		QS     :	BOOL;
		Q0     :	BOOL;
		Q1     :	BOOL;
		Q2     :	BOOL;
		Q3     :	BOOL;
		ERROR  :	BOOL;
		STATUS :	BYTE;

	func_block : FLOW_CONTROL_4;
  END_VAR
	func_block.I0  :=I0  ;
	func_block.I1  :=I1  ;
	func_block.I2  :=I2  ;
	func_block.I3  :=I3  ;
	func_block.PR  :=PR  ;
	func_block.ICE :=ICE ;
	func_block.DIAG:=DIAG;
	func_block.ENQ :=ENQ ;
	func_block.RST :=RST ;
	func_block.TD_WAIT:=TD_WAIT;
	func_block.TD_S   :=TD_S   ;
	func_block.TD_0   :=TD_0   ;
	func_block();
	QS    := func_block.QS    ;
	Q0    := func_block.Q0    ;
	Q1    := func_block.Q1    ;
	Q2    := func_block.Q2    ;
	Q3    := func_block.Q3    ;
	ERROR := func_block.ERROR ;
	STATUS:= func_block.STATUS;

END_PROGRAM

(* ---- lb_claude_assisted_a81a1d0dcc44_0018.st ---- *)
(*
This code implements a randomly grown symbolic expression:

((xor(xor(IN45 & (!(((xor(xor((IN12 | IN39) & (IN49 & IN44), (xor(xor(IN32, IN2), IN29)) | (!(IN23))), !(IN43))) & ((xor(xor(!(IN34), xor(xor(IN7, IN24), IN32)), IN44 & IN23)) & (!(IN26 | IN12)))) & (xor(xor(true, (!(!(IN14))) | IN32), !((IN3 | IN34) & (xor(xor(true, IN16), IN29))))))), (true & (xor(xor(!(IN12), IN38 & ((!(IN22 & IN30)) & ((IN49 & IN6) & (xor(xor(IN28, IN16), IN47))))), IN30))) | (IN20 | (!(!(xor(xor((xor(xor(IN18, IN11), IN44)) | (IN1 | IN1), !(!(IN21))), xor(xor(!(IN27), IN8 | IN35), IN10 | IN21))))))), (IN35 | (!((!(xor(xor(!(IN11), xor(xor(IN5, IN39), IN18)), IN48 | IN49))) & (xor(xor(!(IN2 & IN40), !(IN47 & IN16)), !(xor(xor(IN48, IN6), IN12))))))) & false)) & IN28) | ((!(((((xor(xor(xor(xor(xor(xor(IN26, IN40), IN46), IN25), IN34 & IN49), (!(IN22)) & (!(IN24))), IN22)) & (((IN44 | IN23) & IN20) & (!(IN14 | IN43)))) | IN43) & ((xor(xor(IN5, (xor(xor(IN37, IN49 & IN28), xor(xor(IN22, IN20), IN30))) | ((!(IN46)) | (IN7 | IN28))), (!(IN11 | IN38)) & IN28)) | (!(IN6)))) | (xor(xor(IN22, !((((xor(xor(IN22, IN46), IN13)) | (xor(xor(IN33, IN13), IN13))) & IN3) & (xor(xor((!(IN19)) & (IN23 & IN43), IN9), !(IN47 | IN16))))), xor(xor(((xor(xor(IN41 | IN8, IN31), IN20 | IN5)) & IN33) & (xor(xor(!(IN34), (IN44 | true) & (IN24 | IN13)), IN19)), !(IN24)), !(IN43)))))) & IN28)

*)

FUNCTION_BLOCK F_CollectInput
  VAR_IN_OUT
      Data : ARRAY[1..50] OF BOOL;
  END_VAR
  VAR_INPUT
      TICK  : BOOL := 0;
      IN1   : BOOL := 0;
      IN2   : BOOL := 0;
      IN3   : BOOL := 0;
      IN4   : BOOL := 0;
      IN5   : BOOL := 0;
      RESET : BOOL := FALSE;
  END_VAR
  VAR_OUTPUT
      Finished : BOOL;
  END_VAR
  VAR
      j    : USINT := 1;
      tock : BOOL  := 0;
  END_VAR
  IF NOT RESET AND tock = NOT TICK THEN
      Data[j]   := IN1;
      Data[j+1] := IN2;
      Data[j+2] := IN3;
      Data[j+3] := IN4;
      Data[j+4] := IN5;
      j := j + 5;
      tock := TICK;
  ELSE
      j := 1;
      tock := 0;
  END_IF;
  Finished := (j > 50);
END_FUNCTION_BLOCK

PROGRAM Boiler
  VAR
    Data  : ARRAY[1..50] OF BOOL;
    Ready : BOOL;
    CollectInput : F_CollectInput;
  END_VAR
  VAR
    TICK     AT %IX1.0 : BOOL;
    IN1      AT %IX0.3 : BOOL;
    IN2      AT %IX0.4 : BOOL;
    IN3      AT %IX0.5 : BOOL;
    IN4      AT %IX0.6 : BOOL;
    IN5      AT %IX0.7 : BOOL;
    OutReady AT %QX0.0 : BOOL := FALSE;
    FeedNext AT %QX0.1 : BOOL := FALSE;
    Out      AT %QX0.2 : BOOL;
  END_VAR
  CollectInput(TICK:=TICK, IN1:=IN1, IN2:=IN2, IN3:=IN3, IN4:=IN4, IN5:=IN5);
  Ready := CollectInput.Finished;
  FeedNext := 1;
  IF Ready THEN
    Out := (((((Data[45] AND (NOT ((((((Data[12] OR Data[39]) AND (Data[49] AND Data[44])) XOR (((Data[32] XOR Data[2]) XOR Data[29]) OR (NOT Data[23]))) XOR (NOT Data[43])) AND ((((NOT Data[34]) XOR ((Data[7] XOR Data[24]) XOR Data[32])) XOR (Data[44] AND Data[23])) AND (NOT (Data[26] OR Data[12])))) AND ((TRUE XOR ((NOT (NOT Data[14])) OR Data[32])) XOR (NOT ((Data[3] OR Data[34]) AND ((TRUE XOR Data[16]) XOR Data[29]))))))) XOR ((TRUE AND (((NOT Data[12]) XOR (Data[38] AND ((NOT (Data[22] AND Data[30])) AND ((Data[49] AND Data[6]) AND ((Data[28] XOR Data[16]) XOR Data[47]))))) XOR Data[30])) OR (Data[20] OR (NOT (NOT (((((Data[18] XOR Data[11]) XOR Data[44]) OR (Data[1] OR Data[1])) XOR (NOT (NOT Data[21]))) XOR (((NOT Data[27]) XOR (Data[8] OR Data[35])) XOR (Data[10] OR Data[21])))))))) XOR ((Data[35] OR (NOT ((NOT (((NOT Data[11]) XOR ((Data[5] XOR Data[39]) XOR Data[18])) XOR (Data[48] OR Data[49]))) AND (((NOT (Data[2] AND Data[40])) XOR (NOT (Data[47] AND Data[16]))) XOR (NOT ((Data[48] XOR Data[6]) XOR Data[12])))))) AND FALSE)) AND Data[28]) OR ((NOT ((((((((((Data[26] XOR Data[40]) XOR Data[46]) XOR Data[25]) XOR (Data[34] AND Data[49])) XOR ((NOT Data[22]) AND (NOT Data[24]))) XOR Data[22]) AND (((Data[44] OR Data[23]) AND Data[20]) AND (NOT (Data[14] OR Data[43])))) OR Data[43]) AND (((Data[5] XOR (((Data[37] XOR (Data[49] AND Data[28])) XOR ((Data[22] XOR Data[20]) XOR Data[30])) OR ((NOT Data[46]) OR (Data[7] OR Data[28])))) XOR ((NOT (Data[11] OR Data[38])) AND Data[28])) OR (NOT Data[6]))) OR ((Data[22] XOR (NOT (((((Data[22] XOR Data[46]) XOR Data[13]) OR ((Data[33] XOR Data[13]) XOR Data[13])) AND Data[3]) AND ((((NOT Data[19]) AND (Data[23] AND Data[43])) XOR Data[9]) XOR (NOT (Data[47] OR Data[16])))))) XOR (((((((Data[41] OR Data[8]) XOR Data[31]) XOR (Data[20] OR Data[5])) AND Data[33]) AND (((NOT Data[34]) XOR ((Data[44] OR TRUE) AND (Data[24] OR Data[13]))) XOR Data[19])) XOR (NOT Data[24])) XOR (NOT Data[43]))))) AND Data[28]));
    IF Ready THEN
        OutReady := 0;
    ELSE
        OutReady := 1;
    END_IF;
    CollectInput(RESET:=TRUE);
  END_IF;
END_PROGRAM

CONFIGURATION Config0
  RESOURCE Res0 ON PLC
    TASK task0(INTERVAL := T#20ms,PRIORITY := 0);
    PROGRAM instance0 WITH task0 : Boiler;
  END_RESOURCE
END_CONFIGURATION
